PROGRAM MAIN
VAR
	pbGapMode: BOOL:=FALSE;
	pbTaperMode: BOOL:=FALSE;
	pbSingleCarrierMode: BOOL:=FALSE;
	pbDebugMode:BOOL:=FALSE;
	pbBCGapMode:BOOL:=FALSE;
	fb_led_Show: FB_LedShow;
	btn_reset: BOOL;
	CPMU_PLC_Reset: PLC_Reset;
	d_state: DINT;
	CPMU_PLC_Start: PLC_Start;
	powerStatus:BOOL;

(*TwinSAFE*)
	Safe_run AT%Q*:BOOL;
	Err_Ack AT %Q*:BOOL;
	Estop_RunAndRestart AT %Q*:BOOL;
	AX5805_Error_Ack AT %Q*:BOOL;
	Led_Run  AT %Q*:BOOL;
	Led_Error  AT %Q*:BOOL;

	FB_ERROR AT%I*:BOOL;
	COM_ERROR AT%I*:BOOL;
	//OUT_ERROR AT%I*:BOOL;
	Estop_Out AT%I*:BOOL;

	SafeStatus:INT;
	SafePLCRunOK: BOOL;
	fb_ton: TON;
	fb_ton2: TON;
	fb_ton3: TON;
	fb_ton1: TON;
	fb_ton0: TON;
(*IO*)
	el1808_D1  AT%I* :ARRAY[1..12] OF BOOL;
	el1808_D2  AT%I* :ARRAY[1..4] OF BOOL;
	el1008 AT%I*:BOOL;
	EStopTrig:BOOL;
(*setAxisPosition*)
	SetAxisPosState: INT;
	FB_Set_AxisPosition:FB_SetAxisPosition;
	fb_ton4: TON;
	fb_ton5: TON;
	fb_ton6: TON;
	SetAxisPositionDone: BOOL;
	//
	SetPhaseUpperAxisPosState: INT;
	FB_Set_PhaseUpperAxisPosition:FB_SetPhaseUpperAxisPosition;
	fb_ton7: TON;
	fb_ton8: TON;
	fb_ton9: TON;
	SetPhaseUpperAxisPositionDone: BOOL;
	//
	SetPhaseLowerAxisPosState: INT;
	FB_Set_PhaseLowerAxisPosition:FB_SetPhaseLowerAxisPosition;
	fb_ton10: TON;
	fb_ton11: TON;
	fb_ton12: TON;
	SetPhaseLowerAxisPositionDone: BOOL;
	i: INT;
	j: INT;

(****RS232***)
	fbEL6001	: FB_SerialCom;
	moveDoneLeftTop: BOOL;
	moveDoneRightTop: BOOL;
	moveDoneLeftBottom: BOOL;
	moveDoneRightBottom: BOOL;

(*Torque*)
	Torque_LT AT%I*:INT;
	Torque_RT AT%I*:INT;
	Torque_LB AT%I*:INT;
	Torque_RB AT%I*:INT;
	Torque_PU AT%I*:INT;
	Torque_PL AT%I*:INT;
(**)
	btn_setAxisPosition: BOOL;
	ValueSet_LeftTop:LREAL;
	ValueSet_RightTop:LREAL;
	ValueSet_LeftBottom:LREAL;
	ValueSet_RightBottom:LREAL;
	btn_setPhaseUpperAxisPosition: BOOL;
	PhaseUpperSetValue: LREAL;
	btn_setPhaseLowerAxisPosition: BOOL;
	PhaseLowerSetValue: LREAL;
(**)
	RestartTC: TC_Restart;
	
(*recipe*)
	RecipeINT:INT;
	RecipeBOOL:BOOL;
	RecipeManCommands: RecipeManCommands;
	SaveParameter : BOOL;  //保存文件
	LoadParameter : BOOL;  //读取文件
	Save_R_TRIG   : R_TRIG;
	Read_R_TRIG   : R_TRIG;
	loadparameterStatus: INT;
	RecipeBOOL2:BOOL;
	ReturnDwordLoad: DWORD;
	InsertionDeviceName:STRING;
(*UserMode*)
	pbUserMode: BOOL:=TRUE;
	EL1904 AT%I* :ARRAY[1..32] OF BOOL;
	setAxisPositionEnable: BOOL;
	setPhaseUpperAxisPositionEnable: BOOL;
	setPhaseLowerAxisPositionEnable: BOOL;
	state_loadParameters: INT;
	state_setLEPosBias: INT;
	//
	PositionBiasSet:BOOL;
	MC_SetLEPosBias_LeftTop:MC_WriteParameter;
	MC_SetLEPosBias_RightTop:MC_WriteParameter;
	MC_SetLEPosBias_LeftBottom:MC_WriteParameter;
	MC_SetLEPosBias_RightBottom:MC_WriteParameter;
	MC_SetLEPosBias_PhaseUpper:MC_WriteParameter;
	MC_SetLEPosBias_PhaseLower:MC_WriteParameter;
	PositionBias_LeftTop: LREAL:=10.1;
	PositionBias_RightTop: LREAL:=10.2;
	PositionBias_LeftBottom: LREAL:=10.3;
	PositionBias_RightBottom: LREAL:=10.4;
	PositionBias_PhaseUpper: LREAL:=10.3;
	PositionBias_PhaseLower: LREAL:=10.4;
	
	LoadLEPB_R_TRIG: R_TRIG;
	PositionBiasTON: TON;
	
	//
	OPC_TEST_Bi:BOOL:=TRUE; (*~ (OPC:1:available for OPC Clients) *)
	OPC_TEST_Bi2:BOOL;(*~ (OPC:1:available for OPC Clients) *)
	//
	HasTemperatureSensorOrNot:BOOL;//Only IVU or CPMU
	(*Sensor Reading*)
	Sensor_Reading_1 AT %I*:ARRAY[0..3] OF BYTE;
	Sensor_Reading_2 AT %I*:ARRAY[0..3] OF BYTE;
	Sensor_Reading_3 AT %I*:ARRAY[0..3] OF BYTE;
	Sensor_Reading_4 AT %I*:ARRAY[0..3] OF BYTE;
	Sensor_Reading_5 AT %I*:ARRAY[0..3] OF BYTE;
	Sensor_Reading_6 AT %I*:ARRAY[0..3] OF BYTE;
	Sensor_Reading_7 AT %I*:ARRAY[0..3] OF BYTE;
	Sensor_Reading_8 AT %I*:ARRAY[0..3] OF BYTE;
	Sensor_Reading_DpState AT %I*:USINT;
	Sensor_Reading_ExtDiagFlag AT %I*:BOOL;
	TemperatureSensors_1:LREAL;
	TemperatureSensors_2:LREAL;
	TemperatureSensors_3:LREAL;
	TemperatureSensors_4:LREAL;
	TemperatureSensors_5:LREAL;
	TemperatureSensors_6:LREAL;
	TemperatureSensors_7:LREAL;
	TemperatureSensors_8:LREAL;
	dut_sensor_datas_1:DUT_SENSOR_DATAS_1;
	dut_sensor_datas_2:DUT_SENSOR_DATAS_2;
	dut_sensor_datas_3:DUT_SENSOR_DATAS_3;
	dut_sensor_datas_4:DUT_SENSOR_DATAS_4;
	dut_sensor_datas_5:DUT_SENSOR_DATAS_5;
	dut_sensor_datas_6:DUT_SENSOR_DATAS_6;
	dut_sensor_datas_7:DUT_SENSOR_DATAS_7;
	dut_sensor_datas_8:DUT_SENSOR_DATAS_8;
	//
	temperature_gradient_2_To_1:LREAL;
	temperature_gradient_3_To_2:LREAL;
	temperature_gradient_5_To_4:LREAL;
	temperature_gradient_6_To_5:LREAL;
	temperature_gradient_max:LREAL;
	//
	temperature_average:LREAL;
	A_SetLinearEncoderPositionBias_Enable: BOOL;
	
		//
	temperatureStatus:INT;//0：有传感器度数错误；1:常温；2:低温；3:常温和低温中间态
	CryogenicTemperatureThreshold:LREAL:=80;//80K以下归划分为低温
	RoomTemperatureThreshold:LREAL:=293;//293K以上划分为常温
	//CPMU cryogenix ON/FF
	CryogenicCompensationOn:BOOL;
	CryogenicCompensationConditionsReady:BOOL;
	CryogenicCompensation_LeftTop:LREAL;
	CryogenicCompensation_RightTop:LREAL;
	CryogenicCompensation_LeftBottom:LREAL;
	CryogenicCompensation_RightBottom:LREAL;
	CryogenicCompensationDone: BOOL;
	
	(**)
	bDriveDiagMessageAndNumber  : BOOL;
	m_GetDriveStatusState:INT;
	GetDriveStatusStateDone:BOOL;
	GetDriveStatusStateError:BOOL;
	//	
	fb_SoEReadDiagMessage_LeftTop: FB_SoEReadDiagMessage;
	fb_SoEReadDiagMessage_RightTop: FB_SoEReadDiagMessage;
	fb_SoEReadDiagMessage_LeftBottom: FB_SoEReadDiagMessage;
	fb_SoEReadDiagMessage_RightBottom: FB_SoEReadDiagMessage;
	fb_SoEReadDiagMessage_PhaseUpper: FB_SoEReadDiagMessage;
	fb_SoEReadDiagMessage_PhaseLower: FB_SoEReadDiagMessage;
	DriveDiagMessage_LeftTop:STRING;
	DriveDiagMessage_RightTop:STRING;
	DriveDiagMessage_LeftBottom:STRING;
	DriveDiagMessage_RightBottom:STRING;
	DriveDiagMessage_PhaseUpper:STRING;
	DriveDiagMessage_PhaseLower:STRING;
	//
	FB_SoEReadDiagNumber_LeftTop: FB_SoEReadDiagNumber;
	FB_SoEReadDiagNumber_RightTop: FB_SoEReadDiagNumber;
	FB_SoEReadDiagNumber_LeftBottom: FB_SoEReadDiagNumber;
	FB_SoEReadDiagNumber_RightBottom: FB_SoEReadDiagNumber;
	FB_SoEReadDiagNumber_PhaseUpper: FB_SoEReadDiagNumber;
	FB_SoEReadDiagNumber_PhaseLower: FB_SoEReadDiagNumber;
	DriveDiagNumber_LeftTop:UDINT;
	DriveDiagNumber_RightTop:UDINT;
	DriveDiagNumber_LeftBottom:UDINT;
	DriveDiagNumber_RightBottom:UDINT;
	DriveDiagNumber_PhaseUpper:UDINT;
	DriveDiagNumber_PhaseLower:UDINT;
	bReloadDriveDiagMessageAndNumber: BOOL;
	
	(*load IOC*)
	bExe_load_Prog: BOOL;
	NT_StartProcess_Load: NT_StartProcess;
	Exe_load_step: UINT;
	R_TRIG_ExeLoad: R_TRIG;
	Exe_Load_Done:BOOL;
	(*kill IOC*)
	bExe_Kill_Prog: BOOL;
	NT_StartProcess_Kill: NT_StartProcess;
	Exe_kill_step: UINT;
	R_TRIG_Exekill: R_TRIG;
	Exe_Kill_Done:BOOL;
	LoadOpcIocTON:TON;
	
	GetDriveStatusTON:TON;
	
	//
	//more parameters get:gear;feedback2 direction 
	//
	//GetMoreDriveStatus_FunctionON:BOOL:=TRUE;
	GetDriveStatusTON2: TON;
	//GearNumerator,st182
	st_p182_LeftTop:ST_P182;
	FB_SoERead_GearNumerator_LeftTop: FB_SoERead;
	st_p182_RightTop:ST_P182;
	FB_SoERead_GearNumerator_RightTop: FB_SoERead;
	st_p182_LeftBottom:ST_P182;
	FB_SoERead_GearNumerator_LeftBottom: FB_SoERead;
	st_p182_RightBottom:ST_P182;
	FB_SoERead_GearNumerator_RightBottom: FB_SoERead;
	st_p182_PhaseUpper:ST_P182;
	FB_SoERead_GearNumerator_PhaseUpper: FB_SoERead;
	st_p182_PhaseLower:ST_P182;
	FB_SoERead_GearNumerator_PhaseLower: FB_SoERead;
	GearNumeratorGet_LeftTop:UDINT;
	GearNumeratorGet_RightTop:UDINT;
	GearNumeratorGet_LeftBottom:UDINT;
	GearNumeratorGet_RightBottom:UDINT;
	GearNumeratorGet_PhaseUpper:UDINT;
	GearNumeratorGet_PhaseLower:UDINT;
	GearNumeratorConfigured_LeftTop:UDINT;
	GearNumeratorConfigured_RightTop:UDINT;
	GearNumeratorConfigured_LeftBottom:UDINT;
	GearNumeratorConfigured_RightBottom:UDINT;
	GearNumeratorConfigured_PhaseUpper:UDINT;
	GearNumeratorConfigured_PhaseLower:UDINT;
	//GearDenominator,st183
	st_p183_LeftTop:ST_P183;
	FB_SoERead_GearDenominator_LeftTop: FB_SoERead;
	st_p183_RightTop:ST_P183;
	FB_SoERead_GearDenominator_RightTop: FB_SoERead;
	st_p183_LeftBottom:ST_P183;
	FB_SoERead_GearDenominator_LeftBottom: FB_SoERead;
	st_p183_RightBottom:ST_P183;
	FB_SoERead_GearDenominator_RightBottom: FB_SoERead;
	st_p183_PhaseUpper:ST_P183;
	FB_SoERead_GearDenominator_PhaseUpper: FB_SoERead;
	st_p183_PhaseLower:ST_P183;
	FB_SoERead_GearDenominator_PhaseLower: FB_SoERead;
	GearDenominatorGet_LeftTop:UDINT;
	GearDenominatorGet_RightTop:UDINT;
	GearDenominatorGet_LeftBottom:UDINT;
	GearDenominatorGet_RightBottom:UDINT;
	GearDenominatorGet_PhaseUpper:UDINT;
	GearDenominatorGet_PhaseLower:UDINT;
	GearDenominatorConfigured_LeftTop:UDINT;
	GearDenominatorConfigured_RightTop:UDINT;
	GearDenominatorConfigured_LeftBottom:UDINT;
	GearDenominatorConfigured_RightBottom:UDINT;
	GearDenominatorConfigured_PhaseUpper:UDINT;
	GearDenominatorConfigured_PhaseLower:UDINT;
	//Feedback2direction,st180
	st_p180_LeftTop:ST_P180;
	FB_SoERead_Feedback2direction_LeftTop: FB_SoERead;
	st_p180_RightTop:ST_P180;
	FB_SoERead_Feedback2direction_RightTop: FB_SoERead;
	st_p180_LeftBottom:ST_P180;
	FB_SoERead_Feedback2direction_LeftBottom: FB_SoERead;
	st_p180_RightBottom:ST_P180;
	FB_SoERead_Feedback2direction_RightBottom: FB_SoERead;
	st_p180_PhaseUpper:ST_P180;
	FB_SoERead_Feedback2direction_PhaseUpper: FB_SoERead;
	st_p180_PhaseLower:ST_P180;
	FB_SoERead_Feedback2direction_PhaseLower: FB_SoERead;
	Feedback2directionGet_LeftTop:UINT;
	Feedback2directionGet_RightTop:UINT;
	Feedback2directionGet_LeftBottom:UINT;
	Feedback2directionGet_RightBottom:UINT;
	Feedback2directionGet_PhaseUpper:UINT;
	Feedback2directionGet_PhaseLower:UINT;
	Feedback2directionConfigured_LeftTop:UINT;
	Feedback2directionConfigured_RightTop:UINT;
	Feedback2directionConfigured_LeftBottom:UINT;
	Feedback2directionConfigured_RightBottom:UINT;
	Feedback2directionConfigured_PhaseUpper:UINT;
	Feedback2directionConfigured_PhaseLower:UINT;
	
	//RestartDrivers
		(*重启驱动器*)
	btn_RestartDriversAll:BOOL;
	btn_RestartDriver1:BOOL;
	btn_RestartDriver2:BOOL;
	btn_RestartDriver3:BOOL;
	btn_RestartDriver4:BOOL;
	btn_RestartDriver5:BOOL;
	btn_RestartDriver6:BOOL;
	btn_RestartDriver7:BOOL;
	btn_RestartDriver8:BOOL;
	Relay_EL2624 AT %Q*:ARRAY[0..7]OF  BOOL;
	RestartDriver_RTRIG:R_TRIG;
	RestartDriver_TON:TON;
	RestartDriver_Triggered:BOOL;
	RestartDriver_State:DINT;
	RestartDriver_Done:BOOL;
	//
	
	//
	//	LEHeartBeatMonitorFunction
	//
	LEHeartBeatMonitorFunctionOn: BOOL;
	LEHeartBeatFirstScan:BOOL;
	LEHeartBeatDeadZone : LREAL := 0; 
	LEHeartBeatAlarmTime : TIME := T#0.1S;
	
    //Pos_LeftTopLin_Last : LREAL; 
	Velo_LeftTopLin_Last : LREAL; 
	Pos_LeftTopMotor_Initial : LREAL; 
    StableTimer_LeftTopLin : TON; 
    StableTime_LeftTopLin : TIME; 
    DeltaVelo_LeftTopLin : LREAL; 
	IsInitialPositionSet_LeftTop: BOOL;
	MotorPosChange_LeftTop: LREAL;
	Threshold_LeftTopMotorPos:LREAL:=0.1;
	Threshold_LeftTopMotorVelo:LREAL:=0.2;
	Alarm_LeftTopLin:BOOL;
	Alarm_LeftTopMotorPos:BOOL;
	Alarm_LeftTopMotorVelo:BOOL;
	
	
	//Pos_RightTopLin_Last : LREAL; 
	Velo_RightTopLin_Last : LREAL; 
	Pos_RightTopMotor_Initial : LREAL; 
    StableTimer_RightTopLin : TON; 
    StableTime_RightTopLin : TIME; 
    DeltaVelo_RightTopLin : LREAL; 
	IsInitialPositionSet_RightTop: BOOL;
	MotorPosChange_RightTop: LREAL; 
	Threshold_RightTopMotorPos:LREAL:=0.1;
	Threshold_RightTopMotorVelo:LREAL:=0.2;
	Alarm_RightTopLin:BOOL;
	Alarm_RightTopMotorPos:BOOL;
	Alarm_RightTopMotorVelo:BOOL;
	
		
    //Pos_LeftBottomLin_Last : LREAL; 
	Velo_LeftBottomLin_Last : LREAL; 
	Pos_LeftBottomMotor_Initial : LREAL; 
    StableTimer_LeftBottomLin : TON; 
    StableTime_LeftBottomLin : TIME; 
    DeltaVelo_LeftBottomLin : LREAL; 
	IsInitialPositionSet_LeftBottom: BOOL;
	MotorPosChange_LeftBottom: LREAL; 
	Threshold_LeftBottomMotorPos:LREAL:=0.1;
	Threshold_LeftBottomMotorVelo:LREAL:=0.2;
	Alarm_LeftBottomLin:BOOL;
	Alarm_LeftBottomMotorPos:BOOL;
	Alarm_LeftBottomMotorVelo:BOOL;
	
	//Pos_RightBottomLin_Last : LREAL; 
	Velo_RightBottomLin_Last : LREAL; 
	Pos_RightBottomMotor_Initial : LREAL; 
    StableTimer_RightBottomLin : TON; 
    StableTime_RightBottomLin : TIME; 
    DeltaVelo_RightBottomLin : LREAL; 
	IsInitialPositionSet_RightBottom: BOOL;
	MotorPosChange_RightBottom: LREAL; 
	Threshold_RightBottomMotorPos:LREAL:=0.1;
	Threshold_RightBottomMotorVelo:LREAL:=0.2;
	Alarm_RightBottomLin:BOOL;
	Alarm_RightBottomMotorPos:BOOL;
	Alarm_RightBottomMotorVelo:BOOL;
	
	//Pos_PhaseUpperLin_Last : LREAL; 
	Velo_PhaseUpperLin_Last : LREAL; 
	Pos_PhaseUpperMotor_Initial : LREAL; 
    StableTimer_PhaseUpperLin : TON; 
    StableTime_PhaseUpperLin : TIME; 
    DeltaVelo_PhaseUpperLin : LREAL; 
	IsInitialPositionSet_PhaseUpper: BOOL;
	MotorPosChange_PhaseUpper: LREAL; 
	Threshold_PhaseUpperMotorPos:LREAL:=0.1;
	Threshold_PhaseUpperMotorVelo:LREAL:=0.2;
	Alarm_PhaseUpperLin:BOOL;
	Alarm_PhaseUpperMotorPos:BOOL;
	Alarm_PhaseUpperMotorVelo:BOOL;
	
	//Pos_PhaseLowerLin_Last : LREAL; 
	Velo_PhaseLowerLin_Last : LREAL; 
	Pos_PhaseLowerMotor_Initial : LREAL; 
    StableTimer_PhaseLowerLin : TON; 
    StableTime_PhaseLowerLin : TIME; 
    DeltaVelo_PhaseLowerLin : LREAL; 
	IsInitialPositionSet_PhaseLower: BOOL;
	MotorPosChange_PhaseLower: LREAL; 
	Threshold_PhaseLowerMotorPos:LREAL:=0.1;
	Threshold_PhaseLowerMotorVelo:LREAL:=0.2;
	Alarm_PhaseLowerLin:BOOL;
	Alarm_PhaseLowerMotorPos:BOOL;
	Alarm_PhaseLowerMotorVelo:BOOL;
	
	(*setAxisPosition*)
	SetMotorAxisPosState: INT;
	FB_Set_MotorAxisPosition:FB_SetMotorAxisPosition;
	fb_ton4_2: TON;
	fb_ton5_2: TON;
	SetMotorAxisPositionDone: BOOL;
	btn_SetMotorAxisPosition: BOOL;	
	(*setAxisPosition-PhaseUpper*)
	SetPhaseUpperMotorAxisPosState: INT;
	FB_Set_PhaseUpperMotorAxisPosition:FB_SetPhaseUpperMotorAxisPosition;
	fb_ton7_2: TON;
	SetPhaseUpperMotorAxisPositionDone: BOOL;
	btn_SetPhaseUpperMotorAxisPosition: BOOL;
	(*setAxisPosition-PhaseLower*)
	SetPhaseLowerMotorAxisPosState: INT;
	FB_Set_PhaseLowerMotorAxisPosition:FB_SetPhaseLowerMotorAxisPosition;
	fb_ton8_2: TON;
	SetPhaseLowerMotorAxisPositionDone: BOOL;
	btn_SetPhaseLowerMotorAxisPosition: BOOL;
	
	
	MonitorMotorAndLEFunctionOn:BOOL:=TRUE;
	
		(*GetMotorTempture*)
	MotorTemperature AT %I*:ARRAY[0..5] OF UINT;
	MotorTemperature_LeftTop:LREAL;
	MotorTemperature_RightTop:LREAL;
	MotorTemperature_LeftBottom:LREAL;
	MotorTemperature_RightBottom:LREAL;
	MotorTemperature_PhaseUpper:LREAL;
	MotorTemperature_PhaseLower:LREAL;

	fbPolar    : FB_PolarizationState;
    stPolarizationParam   : ST_PolarizationParam;
END_VAR

(*MaintenanceMode*)
IF MaintenanceMode THEN
	MaintenanceModeLed:=TRUE;
	RETURN;
ELSE
	MaintenanceModeLed:=FALSE;	
END_IF
(*加载Ricipe参数*)
A_InitRecipeParameters();
(*Restart TwinCAT*)
IF Global_Variables.m_restartTC THEN
(*首先关闭opcIocShell.exe*)	
	bExe_Kill_Prog:=TRUE;
	A_KillOpcIocShellExe();
(*重启TC*)
	IF Exe_Kill_Done THEN
		A_RestartTC();
	END_IF
END_IF
(*******InitAxisParameters*******)
A_InitAxisParameters();
(*******¼à²âÏÞÎ»¿ª¹Ø×´Ì¬£¬·½Ïò¿ØÖÆ&½ô¼±Çé¿öÏÂEStop*******)
A_CheckLimitSwitch();
(*Check Kill Switch*)
A_CheckKillSwitch();
(*******PosDiff¼à¿Ø*******)
A_PosDiffDetectiion();
(*******³õÊ¼»¯SafePlc*******)
IF NOT simulation THEN
A_SafePlcStartInit();
END_IF
(************SetAxisPosition-GAP*********************)
IF  NOT USELinearEncoder AND setAxisPositionEnable AND btn_setAxisPosition THEN
		FB_Set_AxisPosition.ValueSet_LeftTop:=ValueSet_LeftTop;
		FB_Set_AxisPosition.ValueSet_RightTop:=ValueSet_RightTop;
		FB_Set_AxisPosition.ValueSet_LeftBottom:=ValueSet_LeftBottom;
		FB_Set_AxisPosition.ValueSet_RightBottom:=ValueSet_RightBottom;
		A_SetAxisPosition();
END_IF
(************SetAxisPosition-GAP*********************)
IF  NOT USELinearEncoder AND setPhaseUpperAxisPositionEnable AND btn_setPhaseUpperAxisPosition THEN
		FB_Set_PhaseUpperAxisPosition.ValueSet:=PhaseUpperSetValue;
		A_SetPhaseUpperAxisPosition();
END_IF
(************SetAxisPosition-GAP*********************)
IF  NOT USELinearEncoder AND setPhaseLowerAxisPositionEnable AND btn_setPhaseLowerAxisPosition THEN
		FB_Set_PhaseLowerAxisPosition.ValueSet:=PhaseLowerSetValue;
		A_SetPhaseLowerAxisPosition();
END_IF
(*******模式选择******)
IF SafePLCRunOK OR Simulation THEN
	IF pbSingleCarrierMode AND NOT pbTaperMode AND NOT pbGapMode AND NOT pbDebugMode AND NOT pbBCGapMode AND NOT pbUserMode THEN
		SingleCarrierMode();
	ELSIF pbTaperMode  AND NOT pbSingleCarrierMode AND NOT pbGapMode  AND NOT pbDebugMode AND NOT pbBCGapMode AND NOT pbUserMode THEN
		TaperMode();
	ELSIF pbGapMode AND  NOT pbSingleCarrierMode AND NOT pbTaperMode  AND NOT pbDebugMode AND NOT pbBCGapMode AND NOT pbUserMode THEN
		GapMode();
	ELSIF pbDebugMode AND NOT pbGapMode AND NOT pbSingleCarrierMode AND NOT pbTaperMode AND NOT pbBCGapMode  AND NOT pbUserMode THEN
		DebugMode();
	ELSIF pbBCGapMode AND NOT pbGapMode AND NOT pbSingleCarrierMode AND NOT pbTaperMode AND NOT pbDebugMode AND NOT pbUserMode THEN
		BCGapMode();
	ELSIF pbUserMode AND NOT pbGapMode AND NOT pbSingleCarrierMode AND NOT pbTaperMode AND NOT pbDebugMode AND NOT pbBCGapMode THEN
		UserMode();
	END_IF
END_IF
(*******Led Show******)
fb_led_Show();
(*******Check Power status******)
FB_Power(Check:=TRUE);
st_Power:=FB_Power.PowerState;
(******Check Couple Status*****)
FB_CheckCoupleStatus(Check:=TRUE);
st_Couple:=FB_CheckCoupleStatus.CoupleState;

(*********RS232*********************)
BackgroundEL();

(*获取温度传感器数据*)
//A_GetTemperatureSensorsData();

(*设置position bias*)
IF loadParametersDone AND (DriveStatus=1 OR simulation) THEN 
	A_SetLinearEncoderPositionBias();
END_IF
(*检查硬急停状态，包括安全限位、柜门急停、手持急停*)
A_CheckHardwareEmergencyStopStatus();
IF NOT simulation THEN
	A_GetDriverStatus();
END_IF
(*IDControlReady*)
IF ((DriveStatus<>0 AND SafePLCRunOK) OR simulation) AND NOT Error THEN
	IDControlReady:=TRUE;
ELSE
	IDControlReady:=FALSE;
END_IF

(*IOC Start*)
IF SafePLCRunOK OR simulation THEN
	bExe_load_Prog:=TRUE;
	A_LoadOpcIocShellExe();
END_IF

(*RestartDrivers*)
A_RestartDrivers();

(*检查光栅读数是否在范围内*)
A_CheckLinearEncoder();


(*A_LEHeartBeatMonitor*)
IF LEHeartBeatMonitorFunctionOn THEN
	A_LEHeartBeatMonitor();
END_IF
(************SetMotorAxisPosition*********************)
//IDControl 1s after
fb_ton5_2.IN:=IDControlReady;
fb_ton5_2.PT:=T#1S;
fb_ton5_2();
IF fb_ton5_2.Q THEN
	btn_SetMotorAxisPosition:=TRUE;
	btn_SetPhaseUpperMotorAxisPosition:=TRUE;
	btn_SetPhaseLowerMotorAxisPosition:=TRUE;
END_IF
IF  USELinearEncoder AND btn_SetMotorAxisPosition THEN
	IF NOT SetMotorAxisPositionDone THEN
		FB_Set_MotorAxisPosition.ValueSet_LeftTop:=Pos_LeftTopLin;
		FB_Set_MotorAxisPosition.ValueSet_RightTop:=Pos_RightTopLin;
		FB_Set_MotorAxisPosition.ValueSet_LeftBottom:=Pos_LeftBottomLin;
		FB_Set_MotorAxisPosition.ValueSet_RightBottom:=Pos_RightBottomLin;
		A_SetMotorAxisPosition();
	END_IF
END_IF
IF  USELinearEncoder AND btn_SetPhaseUpperMotorAxisPosition THEN
	IF NOT SetPhaseUpperMotorAxisPositionDone THEN
		FB_Set_PhaseUpperMotorAxisPosition.ValueSet:=Pos_PhaseUpperLin;
		A_SetPhaseUpperMotorAxisPosition();
	END_IF
END_IF
IF  USELinearEncoder AND btn_SetPhaseLowerMotorAxisPosition THEN
	IF NOT SetPhaseLowerMotorAxisPositionDone THEN
		FB_Set_PhaseLowerMotorAxisPosition.ValueSet:=Pos_PhaseLowerLin;
		A_SetPhaseLowerMotorAxisPosition();
	END_IF
END_IF
(*A_MonitorMotorAndLE*)
IF MonitorMotorAndLEFunctionOn AND SetMotorAxisPositionDone 
	AND SetPhaseUpperMotorAxisPositionDone AND SetPhaseLowerMotorAxisPositionDone THEN
	A_MonitorMotorAndLE();
END_IF
(*A_CheckMaxVelocity*)
A_CheckMaxVelocity();
(**)
A_GetMotorTemperature();

A_PolarStatus();

ACTION A_CheckHardwareEmergencyStopStatus:
IF 	NOT KS_LeftTop_Far_Contact1 OR
	NOT KS_LeftTop_Far_Contact2 OR
	NOT KS_RightTop_Far_Contact1 OR
	NOT KS_RightTop_Far_Contact2 OR
	NOT KS_LeftBottom_Far_Contact1 OR
	NOT KS_LeftBottom_Far_Contact2 OR
	NOT KS_RightBottom_Far_Contact1 OR
	NOT KS_RightBottom_Far_Contact2 OR
	NOT KS_PhaseUpper_Exit_Contact1 OR
	NOT KS_PhaseUpper_Exit_Contact2 OR
	NOT KS_PhaseLower_Exit_Contact1 OR
	NOT KS_PhaseLower_Exit_Contact2 OR
	
	NOT KS_LeftTop_Near_Contact1 OR
	NOT KS_LeftTop_Near_Contact2 OR
	NOT KS_RightTop_Near_Contact1 OR
	NOT KS_RightTop_Near_Contact2 OR
	NOT KS_LeftBottom_Near_Contact1 OR
	NOT KS_LeftBottom_Near_Contact2 OR
	NOT KS_RightBottom_Near_Contact1 OR
	NOT KS_RightBottom_Near_Contact2 OR
	NOT KS_PhaseUpper_Entrance_Contact1 OR
	NOT KS_PhaseUpper_Entrance_Contact2 OR
	NOT KS_PhaseLower_Entrance_Contact1 OR
	NOT KS_PhaseLower_Entrance_Contact2 OR
(*E-STOP*)
	NOT KS_CabinetEmergency_contact1 OR
	NOT KS_CabinetEmergency_contact2 OR
	NOT KS_handEmergency1_Contact1 OR
	NOT KS_handEmergency1_Contact2 OR
	NOT KS_handEmergency2_Contact1 OR
	NOT KS_handEmergency2_Contact2 OR
	NOT KS_softEmergency2_Contact THEN
	Hardware_EmergencyStop:=FALSE;
ELSE
	Hardware_EmergencyStop:=TRUE;
END_IF
END_ACTION

ACTION A_CheckKillSwitch:
IF simulation THEN
	//EL1904-1
	KS_LeftTop_Far_Contact1:=TRUE;
	KS_LeftTop_Far_Contact2:=TRUE;
	KS_LeftTop_Near_Contact1:=TRUE;
	KS_LeftTop_Near_Contact2:=TRUE;
	//EL1904-2
	KS_RightTop_Far_Contact1:=TRUE;
	KS_RightTop_Far_Contact2:=TRUE;
	KS_RightTop_Near_Contact1:=TRUE;
	KS_RightTop_Near_Contact2:=TRUE;
	//EL1904-3
	KS_LeftBottom_Far_Contact1:=TRUE;
	KS_LeftBottom_Far_Contact2:=TRUE;
	KS_LeftBottom_Near_Contact1:=TRUE;
	KS_LeftBottom_Near_Contact2:=TRUE;
	//EL1904-4
	KS_RightBottom_Far_Contact1:=TRUE;
	KS_RightBottom_Far_Contact2:=TRUE;
	KS_RightBottom_Near_Contact1:=TRUE;
	KS_RightBottom_Near_Contact2:=TRUE;
	//EL1904-5
	KS_PhaseUpper_Exit_Contact1:=TRUE;
	KS_PhaseUpper_Exit_Contact2:=TRUE;
	KS_PhaseUpper_Entrance_Contact1:=TRUE;
	KS_PhaseUpper_Entrance_Contact2:=TRUE;
	//EL1904-6
	KS_PhaseLower_Exit_Contact1:=TRUE;
	KS_PhaseLower_Exit_Contact2:=TRUE;
	KS_PhaseLower_Entrance_Contact1:=TRUE;
	KS_PhaseLower_Entrance_Contact2:=TRUE;
	//EL1904-7
	(*E-STOP*)
	(*柜门急停*)
	KS_CabinetEmergency_contact1:=TRUE;
	KS_CabinetEmergency_contact2:=TRUE;
	(*手持急停-1*)
	KS_handEmergency1_Contact1:=TRUE;
	KS_handEmergency1_Contact2:=TRUE;
	//EL1904-8
	(*手持急停-2*)
	KS_handEmergency2_Contact1:=TRUE;
	KS_handEmergency2_Contact2:=TRUE;
	
	KS_softEmergency2_Contact:=TRUE;
	AX5805_ErrorAsk:=TRUE;
ELSE
	//EL1904-1
	KS_LeftTop_Far_Contact1:=EL1904[1];//c1
	KS_LeftTop_Far_Contact2:=EL1904[2];//c2
	KS_LeftTop_Near_Contact1:=EL1904[3];//c3
	KS_LeftTop_Near_Contact2:=EL1904[4];//c4
	//EL1904-2
	KS_RightTop_Far_Contact1:=EL1904[5];
	KS_RightTop_Far_Contact2:=EL1904[6];
	KS_RightTop_Near_Contact1:=EL1904[7];
	KS_RightTop_Near_Contact2:=EL1904[8];
	//EL1904-3
	KS_LeftBottom_Far_Contact1:=EL1904[9];
	KS_LeftBottom_Far_Contact2:=EL1904[10];
	KS_LeftBottom_Near_Contact1:=EL1904[11];
	KS_LeftBottom_Near_Contact2:=EL1904[12];
	//EL1904-4
	KS_RightBottom_Far_Contact1:=EL1904[13];
	KS_RightBottom_Far_Contact2:=EL1904[14];
	KS_RightBottom_Near_Contact1:=EL1904[15];
	KS_RightBottom_Near_Contact2:=EL1904[16];	
	//EL1904-5
	KS_PhaseUpper_Exit_Contact1:=EL1904[17];
	KS_PhaseUpper_Exit_Contact2:=EL1904[18];
	KS_PhaseUpper_Entrance_Contact1:=EL1904[19];
	KS_PhaseUpper_Entrance_Contact2:=EL1904[20];
	//EL1904-6
	KS_PhaseLower_Exit_Contact1:=EL1904[21];
	KS_PhaseLower_Exit_Contact2:=EL1904[22];
	KS_PhaseLower_Entrance_Contact1:=EL1904[23];
	KS_PhaseLower_Entrance_Contact2:=EL1904[24];
	//EL1904-7
	(*E-STOP*)
	(*柜门急停*)
	KS_CabinetEmergency_contact1:=EL1904[25];
	KS_CabinetEmergency_contact2:=EL1904[26];
	(*手持急停-1*)
	KS_handEmergency1_Contact1:=EL1904[27];
	KS_handEmergency1_Contact2:=EL1904[28];
	//EL1904-8
	(*手持急停-2*)
	KS_handEmergency2_Contact1:=EL1904[29];
	KS_handEmergency2_Contact2:=EL1904[30];
	
	KS_softEmergency2_Contact:=EL1904[31];
	AX5805_ErrorAsk:=EL1904[32];

END_IF
END_ACTION

ACTION A_CheckLimitSwitch:
(*******1.´ÓIO»ñÈ¡ÏÞÎ»×´Ì¬******)
(**)

IF simulation THEN
	(**)
	LS_LeftTop_Far:=TRUE;
	LS_LeftTop_Near:=TRUE;
	LS_RightTop_Far:=TRUE;
	LS_RightTop_Near:=TRUE;
	LS_LeftBottom_Far:=TRUE;
	LS_LeftBottom_Near:=TRUE;
	LS_RightBottom_Far:=TRUE;
	LS_RightBottom_Near:=TRUE;
	LS_PhaseUpper_Entrance:=TRUE;
	LS_PhaseUpper_Exit:=TRUE;
	LS_PhaseLower_Entrance:=TRUE;
	LS_PhaseLower_Exit:=TRUE;
	
ELSE
	LS_LeftTop_Far :=el1808_D1[1];
	LS_LeftTop_Near:=el1808_D1[3];
	LS_RightTop_Far:=el1808_D1[2];
	LS_RightTop_Near:=el1808_D1[4];
	LS_LeftBottom_Far:=el1808_D1[7];
	LS_LeftBottom_Near:=el1808_D1[5];
	LS_RightBottom_Far:=el1808_D1[8];
	LS_RightBottom_Near:=el1808_D1[6];
	LS_PhaseUpper_Entrance:=el1808_D2[1];
	LS_PhaseUpper_Exit:=el1808_D2[2];
	LS_PhaseLower_Entrance:=el1808_D2[3];
	LS_PhaseLower_Exit:=el1808_D2[4];
END_IF


(*
	LS_LeftTop_Top:=TRUE;
	LS_LeftTop_Bottom:=TRUE;
	LS_RightTop_Top:=TRUE;
	LS_RightTop_Bottom:=TRUE;
	LS_LeftBottom_Top:=TRUE;
	LS_LeftBottom_Bottom:=TRUE;
	LS_RightBottom_Top:=TRUE;
	LS_RightBottom_Bottom:=TRUE;
*)
(******2.TopÏÞÎ»»òÕßBottomÏÞÎ»ÓÐÒ»¸ö´¥·¢£¬È«¾Ö±äÁ¿¡£¸øMC_POWERÓÃÓÚ·½Ïò¿ØÖÆ£¬ÓÐÒ»¸öÏÞÎ»Îª´¥·¢ÎªFALSE£¬ÔòUnreach_LSÎªFALSE******)
Unreach_LS_Far:=LS_LeftTop_Far AND LS_RightTop_Far AND LS_LeftBottom_Far AND LS_RightBottom_Far;
Unreach_LS_Near:=LS_LeftTop_Near AND LS_RightTop_Near AND LS_LeftBottom_Near AND LS_RightBottom_Near;
(**************************ÏòTopÔË¶¯Ê±£¬´¥ÅöBottomÏÞÎ»¿ª¹Ø£¬»òÕßÏà·´£¬ESTOP**************************************)
(*
IF LeftTopLin.Status.Moving AND Velo_LeftTopLin>0 THEN
	IF NOT Unreach_LS_Bottom THEN
		Error:=TRUE;
		ErrorID:=61;
		FB_PlcEmergencyStop();
	END_IF
ELSIF LeftTopLin.Status.Moving AND Velo_LeftTopLin<0 THEN
	IF NOT Unreach_LS_Top THEN
		Error:=TRUE;
		ErrorID:=62;
		FB_PlcEmergencyStop();
	END_IF
ELSIF RightTopLin.Status.Moving AND Velo_RightTopLin>0 THEN
	IF NOT Unreach_LS_Bottom THEN
		Error:=TRUE;
		ErrorID:=63;
		FB_PlcEmergencyStop();
	END_IF
ELSIF RightTopLin.Status.Moving AND Velo_RightTopLin<0 THEN
	IF NOT  Unreach_LS_Top THEN
		Error:=TRUE;
		ErrorID:=64;
		FB_PlcEmergencyStop();
	END_IF
ELSIF LeftBottomLin.Status.Moving AND Velo_LeftBottomLin>0 THEN
	IF NOT Unreach_LS_Bottom THEN
		Error:=TRUE;
		ErrorID:=65;
		FB_PlcEmergencyStop();
	END_IF
ELSIF LeftBottomLin.Status.Moving AND Velo_LeftBottomLin<0 THEN
	IF NOT Unreach_LS_Top THEN
		Error:=TRUE;
		ErrorID:=66;
		FB_PlcEmergencyStop();
	END_IF
ELSIF RightBottomLin.Status.Moving AND Velo_RightBottomLin>0 THEN
	IF NOT Unreach_LS_Bottom THEN
		Error:=TRUE;
		ErrorID:=67;
		FB_PlcEmergencyStop();
	END_IF
ELSIF RightBottomLin.Status.Moving AND Velo_RightBottomLin<0 THEN
	IF NOT Unreach_LS_Top THEN
		Error:=TRUE;
		ErrorID:=68;
		FB_PlcEmergencyStop();
	END_IF
END_IF
*)
(*
(******3.ÓÐÒ»¸öÏÞÎ»´¥·¢£¬ delayÊ±¼äºó£¬¼à²âÖáÊÇ·ñÔÚÍ£Ö¹×´Ì¬£¬ÈôÃ»ÓÐ£¬Emergency AND PowerOff******)
IF NOT Unreach_LS_Top OR NOT Unreach_LS_Bottom THEN
	fb_ton.IN:=TRUE;
END_IF
IF fb_ton.Q THEN
	IF LeftTopLin.Status.Moving OR RightTopLin.Status.Moving OR LeftBottomLin.Status.Moving OR RightBottomLin.Status.Moving THEN
		FB_PlcEmergencyStop();
		fb_ton.IN:=FALSE;
		Error:=TRUE;
		EStopTrig:=TRUE;
		ErrorID:=1;
		(*FB_Power_Off(Execute:=TRUE);*)
	END_IF
END_IF

(*******4.µ¥ÖáÉÏÏÂÏÞÎ»¾ùÎªFALSEÊ±£¬ÏÞÎ»´íÎó£¬Emergency*******)
IF (NOT LS_LeftTop_Top AND NOT LS_LeftTop_Bottom) OR  (NOT  LS_RightTop_Top AND NOT LS_RightTop_Bottom)
		OR (NOT LS_LeftBottom_Top AND NOT LS_LeftBottom_Bottom) OR (NOT LS_RightBottom_Top AND NOT LS_RightBottom_Bottom) THEN
	(*FB_Plc_EmergencyStop();*)
	Error:=TRUE;
	EStopTrig:=TRUE;
	ErrorID:=2;
END_IF
*)
END_ACTION

ACTION A_CheckLinearEncoder:
//LE Protection Position
min_UserLEProtectionGapPosition:=min_UserGapPositionNew-min_ThresholdGapSoft2LEProtection;//回程误差有0.1mm
max_UserLEProtectionGapPosition:=max_UserGapPositionNew+max_ThresholdGapSoft2LEProtection;
//如果没有使用光栅、或者光栅参数没设置好，则不检查光栅位置
IF NOT USELinearEncoder OR NOT PositionBiasDone THEN
	RETURN;
END_IF
IF Pos_LeftTopLin <=0 THEN
	ErrorID:=1101;
	Error:=TRUE;
	ErrorDescription:='Pos_LeftTopLin <=0';
	FB_PlcEmergencyStop();
	LED_Error:=TRUE;
END_IF
IF Pos_RightTopLin <=0 THEN
	ErrorID:=1102;
	Error:=TRUE;
	ErrorDescription:='Pos_RightTopLin <=0';
	FB_PlcEmergencyStop();
	LED_Error:=TRUE;
END_IF
IF Pos_LeftBottomLin <=0 THEN
	ErrorID:=1103;
	Error:=TRUE;
	ErrorDescription:='Pos_LeftBottomLin <=0';
	FB_PlcEmergencyStop();
	LED_Error:=TRUE;
END_IF
IF Pos_RightBottomLin <=0 THEN
	ErrorID:=1104;
	Error:=TRUE;
	ErrorDescription:='Pos_RightBottomLin <=0';
	FB_PlcEmergencyStop();
	LED_Error:=TRUE;
END_IF

//
IF Pos_LeftTopLin >max_UserLEProtectionGapPosition/2 THEN
	ErrorID:=1105;
	Error:=TRUE;
	ErrorDescription:='Pos_LeftTopLin >max_UserLEProtectionGapPosition/2';
	FB_PlcEmergencyStop();
	LED_Error:=TRUE;
END_IF
IF Pos_RightTopLin >max_UserLEProtectionGapPosition/2 THEN
	ErrorID:=1106;
	Error:=TRUE;
	ErrorDescription:='Pos_RightTopLin>max_UserLEProtectionGapPosition/2';
	FB_PlcEmergencyStop();
	LED_Error:=TRUE;
END_IF
IF Pos_LeftBottomLin >max_UserLEProtectionGapPosition/2 THEN
	ErrorID:=1107;
	Error:=TRUE;
	ErrorDescription:='Pos_LeftBottomLin >max_UserLEProtectionGapPosition/2';
	FB_PlcEmergencyStop();
	LED_Error:=TRUE;
END_IF
IF Pos_RightBottomLin >max_UserLEProtectionGapPosition/2 THEN
	ErrorID:=1108;
	Error:=TRUE;
	ErrorDescription:='Pos_RightBottomLin >max_UserLEProtectionGapPosition/2';
	FB_PlcEmergencyStop();
	LED_Error:=TRUE;
END_IF


IF Pos_LeftTopLin <min_UserLEProtectionGapPosition/2 THEN
	ErrorID:=1109;
	Error:=TRUE;
	ErrorDescription:='Pos_LeftTopLin <min_UserLEProtectionGapPosition/2';
	FB_PlcEmergencyStop();
	LED_Error:=TRUE;
END_IF
IF Pos_RightTopLin <min_UserLEProtectionGapPosition/2 THEN
	ErrorID:=1110;
	Error:=TRUE;
	ErrorDescription:='Pos_RightTopLin<min_UserLEProtectionGapPosition/2';
	FB_PlcEmergencyStop();
	LED_Error:=TRUE;
END_IF
IF Pos_LeftBottomLin <min_UserLEProtectionGapPosition/2 THEN
	ErrorID:=1111;
	Error:=TRUE;
	ErrorDescription:='Pos_LeftBottomLin <min_UserLEProtectionGapPosition';
	FB_PlcEmergencyStop();
	LED_Error:=TRUE;
END_IF
IF Pos_RightBottomLin <min_UserLEProtectionGapPosition/2 THEN
	ErrorID:=1112;
	Error:=TRUE;
	ErrorDescription:='Pos_RightBottomLin <min_UserLEProtectionGapPosition';
	FB_PlcEmergencyStop();
	LED_Error:=TRUE;
END_IF
//
//PhaseUpper方向
//
min_UserLEProtectionPhaseUpperPosition:=min_UserPhaseUpperPositionNew-min_ThresholdPhaseUpperSoft2LEProtection;//回程误差有0.1mm
max_UserLEProtectionPhaseUpperPosition:=max_UserPhaseUpperPositionNew+max_ThresholdPhaseUpperSoft2LEProtection;
IF Pos_PhaseUpperLin >max_UserLEProtectionPhaseUpperPosition THEN
	ErrorID:=1113;
	Error:=TRUE;
	ErrorDescription:=' Pos_PhaseUpperLin >max_UserLEProtectionPhaseUpperPosition';
	FB_PlcEmergencyStop();
	LED_Error:=TRUE;
END_IF
IF Pos_PhaseUpperLin < min_UserLEProtectionPhaseUpperPosition THEN
	ErrorID:=1114;
	Error:=TRUE;
	ErrorDescription:=' Pos_PhaseUpperLin >< min_UserLEProtectionPhaseUpperPosition';
	FB_PlcEmergencyStop();
	LED_Error:=TRUE;
END_IF
//
//PhaseLower方向
//
min_UserLEProtectionPhaseLowerPosition:=min_UserPhaseLowerPositionNew-min_ThresholdPhaseLowerSoft2LEProtection;//回程误差有0.1mm
max_UserLEProtectionPhaseLowerPosition:=max_UserPhaseLowerPositionNew+max_ThresholdPhaseLowerSoft2LEProtection;
IF Pos_PhaseLowerLin >max_UserLEProtectionPhaseLowerPosition THEN
	ErrorID:=1115;
	Error:=TRUE;
	ErrorDescription:=' Pos_PhaseLowerLin >max_UserLEProtectionPhaseLowerPosition';
	FB_PlcEmergencyStop();
	LED_Error:=TRUE;
END_IF
IF Pos_PhaseLowerLin < min_UserLEProtectionPhaseLowerPosition THEN
	ErrorID:=1116;
	Error:=TRUE;
	ErrorDescription:=' Pos_PhaseLowerLin < min_UserLEProtectionPhaseLowerPosition';
	FB_PlcEmergencyStop();
	LED_Error:=TRUE;
END_IF
END_ACTION

ACTION A_CheckMaxVelocity:
IF NOT USELinearEncoder OR NOT PositionBiasDone OR NOT IDControlReady THEN
	RETURN;
END_IF
IF NOT st_Power THEN
	RETURN;
END_IF
//Monitoring Motor and LE Position/Velocity
MaxVelocityGlobalVelocity:=MAX(max_UserGapVelocityNew,max_UserTaperVelocityNew,UserMode.max_SS_StepVelocity,
			UserMode.Global_ChainProtection_MPS_MoveVelocity,UserMode.Global_ChainProtection_EPS_MoveVelocity);
IF 	ABS(Velo_LeftTopLin) > MaxVelocityGlobalVelocity*1.1/2 THEN
	ErrorID:=7001;
	Error:=TRUE;
	ErrorDescription:='ABS(Velo_LeftTopLin) > MaxVelocityGlobalVelocity*1.1/2';
	FB_PlcEmergencyStop();
	LED_Error:=TRUE;
END_IF
IF 	ABS(Velo_LeftTopMotor) > MaxVelocityGlobalVelocity*1.1/2 THEN
	ErrorID:=7002;
	Error:=TRUE;
	ErrorDescription:='ABS(Velo_LeftTopMotor) > MaxVelocityGlobalVelocity*1.1/2';
	FB_PlcEmergencyStop();
	LED_Error:=TRUE;
END_IF
IF 	ABS(Velo_RightTopLin) > MaxVelocityGlobalVelocity*1.1/2 THEN
	ErrorID:=7003;
	Error:=TRUE;
	ErrorDescription:='ABS(Velo_RightTopLin) > MaxVelocityGlobalVelocity*1.1/2';
	FB_PlcEmergencyStop();
	LED_Error:=TRUE;
END_IF
IF 	ABS(Velo_RightTopMotor) > MaxVelocityGlobalVelocity*1.1/2 THEN
	ErrorID:=7004;
	Error:=TRUE;
	ErrorDescription:='ABS(Velo_RightTopMotor) > MaxVelocityGlobalVelocity*1.1/2';
	FB_PlcEmergencyStop();
	LED_Error:=TRUE;
END_IF
IF 	ABS(Velo_LeftBottomLin) > MaxVelocityGlobalVelocity*1.1/2 THEN
	ErrorID:=7005;
	Error:=TRUE;
	ErrorDescription:='ABS(Velo_LeftBottomLin) > MaxVelocityGlobalVelocity*1.1/2';
	FB_PlcEmergencyStop();
	LED_Error:=TRUE;
END_IF
IF 	ABS(Velo_LeftBottomMotor) > MaxVelocityGlobalVelocity*1.1/2 THEN
	ErrorID:=7006;
	Error:=TRUE;
	ErrorDescription:='ABS(Velo_LeftBottomMotor) > MaxVelocityGlobalVelocity*1.1/2';
	FB_PlcEmergencyStop();
	LED_Error:=TRUE;
END_IF
IF 	ABS(Velo_RightBottomLin) > MaxVelocityGlobalVelocity*1.1/2 THEN
	ErrorID:=7007;
	Error:=TRUE;
	ErrorDescription:='ABS(Velo_RightBottomLin) > MaxVelocityGlobalVelocity*1.1/2';
	FB_PlcEmergencyStop();
	LED_Error:=TRUE;
END_IF
IF 	ABS(Velo_RightBottomMotor) > MaxVelocityGlobalVelocity*1.1/2 THEN
	ErrorID:=7008;
	Error:=TRUE;
	ErrorDescription:='ABS(Velo_RighBottomMotor) > MaxVelocityGlobalVelocity*1.1/2';
	FB_PlcEmergencyStop();
	LED_Error:=TRUE;
END_IF
(*
IF 	ABS(Velo_PhaseUpperLin) > MaxVelocityGlobalVelocity*1.1/2 THEN
	ErrorID:=7005;
	Error:=TRUE;
	ErrorDescription:='ABS(Velo_PhaseUpperLin) > MaxVelocityGlobalVelocity*1.1/2';
	FB_PlcEmergencyStop();
	LED_Error:=TRUE;
END_IF
IF 	ABS(Velo_PhaseUpperMotor) > MaxVelocityGlobalVelocity*1.1/2 THEN
	ErrorID:=7006;
	Error:=TRUE;
	ErrorDescription:='ABS(Velo_PhaseUpperMotor) > MaxVelocityGlobalVelocity*1.1/2';
	FB_PlcEmergencyStop();
	LED_Error:=TRUE;
END_IF
IF 	ABS(Velo_PhaseLowerLin) > MaxVelocityGlobalVelocity*1.1/2 THEN
	ErrorID:=7007;
	Error:=TRUE;
	ErrorDescription:='ABS(Velo_PhaseLowerLin) > MaxVelocityGlobalVelocity*1.1/2';
	FB_PlcEmergencyStop();
	LED_Error:=TRUE;
END_IF
IF 	ABS(Velo_PhaseLowerMotor) > MaxVelocityGlobalVelocity*1.1/2 THEN
	ErrorID:=7008;
	Error:=TRUE;
	ErrorDescription:='ABS(Velo_RighBottomMotor) > MaxVelocityGlobalVelocity*1.1/2';
	FB_PlcEmergencyStop();
	LED_Error:=TRUE;
END_IF
*)
END_ACTION

ACTION A_GetDriverStatus:
//
//DriveMessage/Drive Number/Gear number/feedback2 direction
//
IF bReloadDriveDiagMessageAndNumber THEN
	m_GetDriveStatusState:=0;
	bReloadDriveDiagMessageAndNumber:=FALSE;
END_IF
GetDriveStatusTON(PT:=T#1S);
GetDriveStatusTON2(PT:=T#0.1S);
A_GetDriverStatusMC();
CASE m_GetDriveStatusState OF
	0:
		GetDriveStatusTON.IN:=TRUE;
		m_GetDriveStatusState:=1;
	1:
		IF GetDriveStatusTON.Q THEN
			bDriveDiagMessageAndNumber:=TRUE;
			m_GetDriveStatusState:=2;
		END_IF
	2:
		GetDriveStatusTON.IN:=FALSE;
		DriveDiagMessage_LeftTop:=fb_SoEReadDiagMessage_LeftTop.sDiagMessage.strData;
		DriveDiagMessage_RightTop:=fb_SoEReadDiagMessage_RightTop.sDiagMessage.strData;
		DriveDiagMessage_LeftBottom:=fb_SoEReadDiagMessage_LeftBottom.sDiagMessage.strData;
		DriveDiagMessage_RightBottom:=fb_SoEReadDiagMessage_RightBottom.sDiagMessage.strData;
		DriveDiagMessage_PhaseUpper:=fb_SoEReadDiagMessage_PhaseUpper.sDiagMessage.strData;
		DriveDiagMessage_PhaseLower:=fb_SoEReadDiagMessage_PhaseLower.sDiagMessage.strData;
		//
		DriveDiagNumber_LeftTop:=FB_SoEReadDiagNumber_LeftTop.iDiagNumber;
		DriveDiagNumber_RightTop:=FB_SoEReadDiagNumber_RightTop.iDiagNumber;
		DriveDiagNumber_LeftBottom:=FB_SoEReadDiagNumber_LeftBottom.iDiagNumber;
		DriveDiagNumber_RightBottom:=FB_SoEReadDiagNumber_RightBottom.iDiagNumber;
		DriveDiagNumber_PhaseUpper:=FB_SoEReadDiagNumber_PhaseUpper.iDiagNumber;
		DriveDiagNumber_PhaseLower:=FB_SoEReadDiagNumber_PhaseLower.iDiagNumber;
		//
		GearNumeratorGet_LeftTop:=st_p182_LeftTop.Feedback_2_geat_numerator;
		GearNumeratorGet_RightTop:=st_p182_RightTop.Feedback_2_geat_numerator;
		GearNumeratorGet_LeftBottom:=st_p182_LeftBottom.Feedback_2_geat_numerator;
		GearNumeratorGet_RightBottom:=st_p182_RightBottom.Feedback_2_geat_numerator;
		GearNumeratorGet_PhaseUpper:=st_p182_PhaseUpper.Feedback_2_geat_numerator;
		GearNumeratorGet_PhaseLower:=st_p182_PhaseLower.Feedback_2_geat_numerator;
		//
		GearDenominatorGet_LeftTop:=st_p183_LeftTop.Feedback_2_geat_denominator;
		GearDenominatorGet_RightTop:=st_p183_RightTop.Feedback_2_geat_denominator;
		GearDenominatorGet_LeftBottom:=st_p183_LeftBottom.Feedback_2_geat_denominator;
		GearDenominatorGet_RightBottom:=st_p183_RightBottom.Feedback_2_geat_denominator;
		GearDenominatorGet_PhaseUpper:=st_p183_PhaseUpper.Feedback_2_geat_denominator;
		GearDenominatorGet_PhaseLower:=st_p183_PhaseLower.Feedback_2_geat_denominator;
		//
		Feedback2directionGet_LeftTop:=st_p180_LeftTop.Feedback_direction;
		Feedback2directionGet_RightTop:=st_p180_RightTop.Feedback_direction;
		Feedback2directionGet_LeftBottom:=st_p180_LeftBottom.Feedback_direction;
		Feedback2directionGet_RightBottom:=st_p180_RightBottom.Feedback_direction;
		Feedback2directionGet_PhaseUpper:=st_p180_PhaseUpper.Feedback_direction;
		Feedback2directionGet_PhaseLower:=st_p180_PhaseLower.Feedback_direction;
		//
		IF 	NOT fb_SoEReadDiagMessage_LeftTop.bBusy
			AND NOT fb_SoEReadDiagMessage_RightTop.bBusy
			AND NOT fb_SoEReadDiagMessage_LeftBottom.bBusy
			AND NOT fb_SoEReadDiagMessage_RightBottom.bBusy 
			AND NOT fb_SoEReadDiagMessage_PhaseUpper.bBusy
			AND NOT fb_SoEReadDiagMessage_PhaseLower.bBusy 
			AND NOT FB_SoEReadDiagNumber_LeftTop.bBusy
			AND NOT FB_SoEReadDiagNumber_RightTop.bBusy
			AND NOT FB_SoEReadDiagNumber_LeftBottom.bBusy
			AND NOT FB_SoEReadDiagNumber_RightBottom.bBusy 
			AND NOT FB_SoEReadDiagNumber_PhaseUpper.bBusy
			AND NOT FB_SoEReadDiagNumber_PhaseLower.bBusy 
			AND NOT FB_SoERead_GearNumerator_LeftTop.bBusy 
			AND NOT FB_SoERead_GearNumerator_RightTop.bBusy 
			AND NOT FB_SoERead_GearNumerator_LeftBottom.bBusy 
			AND NOT FB_SoERead_GearNumerator_RightBottom.bBusy 
			AND NOT FB_SoERead_GearNumerator_PhaseUpper.bBusy 
			AND NOT FB_SoERead_GearNumerator_PhaseLower.bBusy 
			AND NOT FB_SoERead_GearDenominator_LeftTop.bBusy 
			AND NOT FB_SoERead_GearDenominator_RightTop.bBusy 
			AND NOT FB_SoERead_GearDenominator_LeftBottom.bBusy 
			AND NOT FB_SoERead_GearDenominator_RightBottom.bBusy 
			AND NOT FB_SoERead_GearDenominator_PhaseUpper.bBusy 
			AND NOT FB_SoERead_GearDenominator_PhaseLower.bBusy 
			AND NOT FB_SoERead_Feedback2direction_LeftTop.bBusy 
			AND NOT FB_SoERead_Feedback2direction_RightTop.bBusy  
			AND NOT FB_SoERead_Feedback2direction_LeftBottom.bBusy 
			AND NOT FB_SoERead_Feedback2direction_RightBottom.bBusy
			AND NOT FB_SoERead_Feedback2direction_PhaseUpper.bBusy 
			AND NOT FB_SoERead_Feedback2direction_PhaseLower.bBusy	THEN
				GetDriveStatusTON2.IN:=TRUE;
				IF GetDriveStatusTON2.Q THEN
					m_GetDriveStatusState:=88;
				END_IF
		END_IF
		IF 	fb_SoEReadDiagMessage_LeftTop.bError
			OR fb_SoEReadDiagMessage_RightTop.bError
			OR fb_SoEReadDiagMessage_LeftBottom.bError
			OR fb_SoEReadDiagMessage_RightBottom.bError
			OR fb_SoEReadDiagMessage_PhaseUpper.bError
			OR fb_SoEReadDiagMessage_PhaseLower.bError
			OR FB_SoEReadDiagNumber_LeftTop.bError
			OR FB_SoEReadDiagNumber_RightTop.bError
			OR FB_SoEReadDiagNumber_LeftBottom.bError
			OR FB_SoEReadDiagNumber_RightBottom.bError 
			OR FB_SoEReadDiagNumber_PhaseUpper.bError
			OR FB_SoEReadDiagNumber_PhaseLower.bError 
			OR FB_SoERead_GearNumerator_LeftTop.bError 
			OR FB_SoERead_GearNumerator_RightTop.bError 
			OR FB_SoERead_GearNumerator_LeftBottom.bError 
			OR FB_SoERead_GearNumerator_RightBottom.bError 
			OR FB_SoERead_GearNumerator_PhaseUpper.bError 
			OR FB_SoERead_GearNumerator_PhaseLower.bError 
			OR FB_SoERead_GearDenominator_LeftTop.bError 
			OR FB_SoERead_GearDenominator_RightTop.bError 
			OR FB_SoERead_GearDenominator_LeftBottom.bError 
			OR FB_SoERead_GearDenominator_RightBottom.bError 
			OR FB_SoERead_GearDenominator_PhaseUpper.bError 
			OR FB_SoERead_GearDenominator_PhaseLower.bError 
			OR FB_SoERead_Feedback2direction_LeftTop.bError 
			OR FB_SoERead_Feedback2direction_RightTop.bError 
			OR FB_SoERead_Feedback2direction_LeftBottom.bError 
			OR FB_SoERead_Feedback2direction_RightBottom.bError 
			OR FB_SoERead_Feedback2direction_PhaseUpper.bError 
			OR FB_SoERead_Feedback2direction_PhaseLower.bError 
		THEN
			m_GetDriveStatusState:=-100;
		END_IF
		
	88:
		bDriveDiagMessageAndNumber:=FALSE;
		A_GetDriverStatusMC();
		GetDriveStatusStateDone:=TRUE;
		GetDriveStatusStateError:=FALSE;
		//
		(*Drive Status*)
		//D012, Axis state machine: Control and power section ready,53266
		IF DriveDiagNumber_LeftTop=16#D012 AND DriveDiagNumber_RightTop=16#D012			
			AND DriveDiagNumber_LeftBottom=16#D012 AND DriveDiagNumber_RightBottom=16#D012
			AND DriveDiagNumber_PhaseUpper=16#D012 AND DriveDiagNumber_PhaseLower=16#D012 THEN
			DriveStatus:=1;
		//D013, Axis state machine: Axis in operation,53267
		ELSIF DriveDiagNumber_LeftTop=16#D013 AND DriveDiagNumber_RightTop=16#D013
			AND DriveDiagNumber_LeftBottom=16#D013 AND DriveDiagNumber_RightBottom=16#D013
			AND DriveDiagNumber_PhaseUpper=16#D013 AND DriveDiagNumber_PhaseLower=16#D013 THEN
			DriveStatus:=2;
		//D014，Axis state machine: Axis halt.53266和53267中间会经历这么一个状态，算正常状态
		ELSIF DriveDiagNumber_LeftTop=16#D014 AND DriveDiagNumber_RightTop=16#D014
			AND DriveDiagNumber_LeftBottom=16#D014 AND DriveDiagNumber_RightBottom=16#D014
			AND DriveDiagNumber_PhaseUpper=16#D014 AND DriveDiagNumber_PhaseLower=16#D014 THEN
			DriveStatus:=3;
		ELSE
			DriveStatus:=0;
		END_IF
		//
		//
		//	//check statusGet and status configured
		IF 	GearNumeratorGet_LeftTop<>GearNumeratorConfigured_LeftTop 
			OR GearNumeratorGet_RightTop<>GearNumeratorConfigured_RightTop
			OR GearNumeratorGet_LeftBottom<>GearNumeratorConfigured_LeftBottom 
			OR GearNumeratorGet_RightBottom<>GearNumeratorConfigured_RightBottom
			OR GearNumeratorGet_PhaseUpper<>GearNumeratorConfigured_PhaseUpper 
			OR GearNumeratorGet_PhaseLower<>GearNumeratorConfigured_PhaseLower
			OR GearDenominatorGet_LeftTop<>GearDenominatorConfigured_LeftTop 
			OR GearDenominatorGet_RightTop<>GearDenominatorConfigured_RightTop
			OR GearDenominatorGet_LeftBottom<>GearDenominatorConfigured_LeftBottom 
			OR GearDenominatorGet_RightBottom<>GearDenominatorConfigured_RightBottom
			OR GearDenominatorGet_PhaseUpper<>GearDenominatorConfigured_PhaseUpper 
			OR GearDenominatorGet_PhaseLower<>GearDenominatorConfigured_PhaseLower THEN
				bDriveDiagMessageAndNumber:=FALSE;
				A_GetDriverStatusMC();
				GetDriveStatusStateDone:=FALSE;
				GetDriveStatusStateError:=TRUE;
				Error:=TRUE;
				ErrorId:=1302;
				ErrorDescription:='gearParameters Error';
				Plc_EmergencyStop:=FALSE;
		END_IF
		IF USELinearEncoder THEN
			IF 	Feedback2directionGet_LeftTop<>Feedback2directionConfigured_LeftTop 
				OR Feedback2directionGet_RightTop<>Feedback2directionConfigured_RightTop
				OR Feedback2directionGet_LeftBottom<>Feedback2directionConfigured_LeftBottom 
				OR Feedback2directionGet_RightBottom<Feedback2directionConfigured_RightBottom 
				OR Feedback2directionGet_PhaseUpper<>Feedback2directionConfigured_PhaseUpper 
				OR Feedback2directionGet_PhaseLower<Feedback2directionConfigured_PhaseLower THEN
					bDriveDiagMessageAndNumber:=FALSE;
					A_GetDriverStatusMC();
					GetDriveStatusStateDone:=FALSE;
					GetDriveStatusStateError:=TRUE;
					Error:=TRUE;
					ErrorId:=1303;
					ErrorDescription:='fb2direction Error';
					Plc_EmergencyStop:=FALSE;
			END_IF 
		END_IF
		m_GetDriveStatusState:=0;
	-100:
		bDriveDiagMessageAndNumber:=FALSE;
		A_GetDriverStatusMC();
		GetDriveStatusStateDone:=FALSE;
		GetDriveStatusStateError:=TRUE;
		Error:=TRUE;
		ErrorId:=1301;
		ErrorDescription:='GetDriveStatusStateError';
END_CASE
END_ACTION

ACTION A_GetDriverStatusMC:
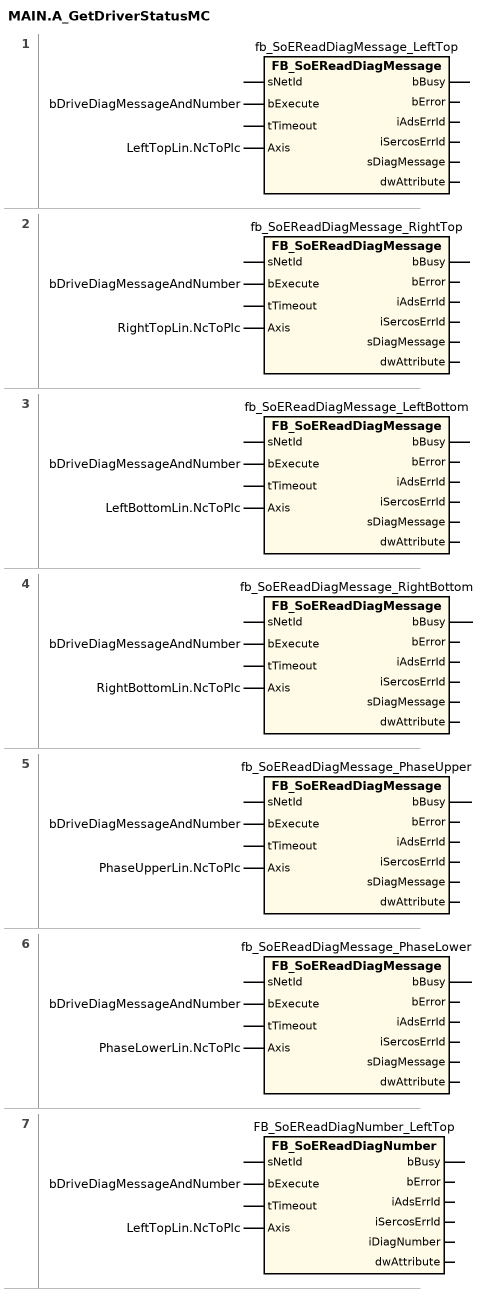
// NETWORK 1
fb_SoEReadDiagMessage_LeftTop(bExecute := bDriveDiagMessageAndNumber, Axis := LeftTopLin.NcToPlc); // FB_SoEReadDiagMessage

// NETWORK 2
fb_SoEReadDiagMessage_RightTop(bExecute := bDriveDiagMessageAndNumber, Axis := RightTopLin.NcToPlc); // FB_SoEReadDiagMessage

// NETWORK 3
fb_SoEReadDiagMessage_LeftBottom(bExecute := bDriveDiagMessageAndNumber, Axis := LeftBottomLin.NcToPlc); // FB_SoEReadDiagMessage

// NETWORK 4
fb_SoEReadDiagMessage_RightBottom(bExecute := bDriveDiagMessageAndNumber, Axis := RightBottomLin.NcToPlc); // FB_SoEReadDiagMessage

// NETWORK 5
fb_SoEReadDiagMessage_PhaseUpper(bExecute := bDriveDiagMessageAndNumber, Axis := PhaseUpperLin.NcToPlc); // FB_SoEReadDiagMessage

// NETWORK 6
fb_SoEReadDiagMessage_PhaseLower(bExecute := bDriveDiagMessageAndNumber, Axis := PhaseLowerLin.NcToPlc); // FB_SoEReadDiagMessage

// NETWORK 7
FB_SoEReadDiagNumber_LeftTop(bExecute := bDriveDiagMessageAndNumber, Axis := LeftTopLin.NcToPlc); // FB_SoEReadDiagNumber

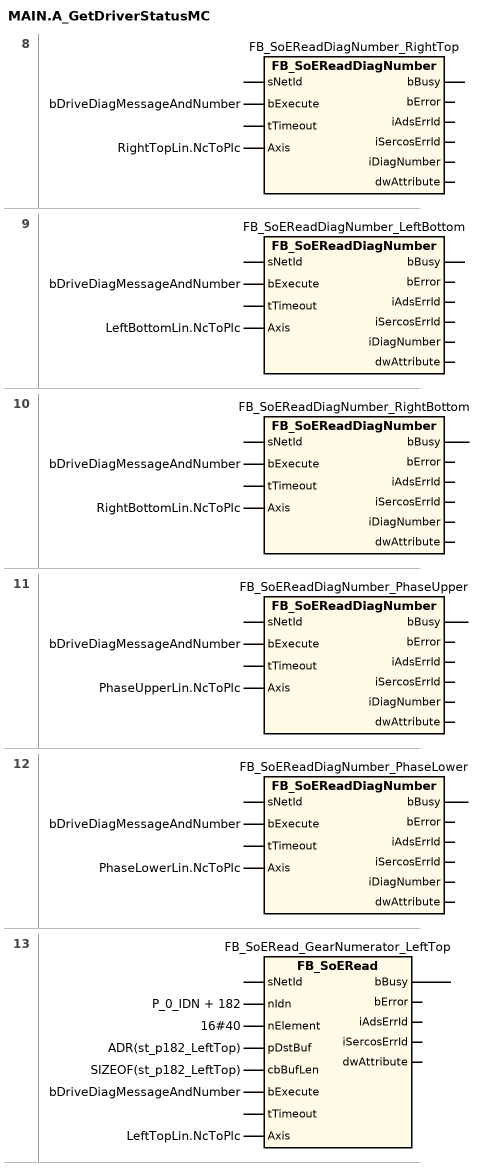
// NETWORK 8
FB_SoEReadDiagNumber_RightTop(bExecute := bDriveDiagMessageAndNumber, Axis := RightTopLin.NcToPlc); // FB_SoEReadDiagNumber

// NETWORK 9
FB_SoEReadDiagNumber_LeftBottom(bExecute := bDriveDiagMessageAndNumber, Axis := LeftBottomLin.NcToPlc); // FB_SoEReadDiagNumber

// NETWORK 10
FB_SoEReadDiagNumber_RightBottom(bExecute := bDriveDiagMessageAndNumber, Axis := RightBottomLin.NcToPlc); // FB_SoEReadDiagNumber

// NETWORK 11
FB_SoEReadDiagNumber_PhaseUpper(bExecute := bDriveDiagMessageAndNumber, Axis := PhaseUpperLin.NcToPlc); // FB_SoEReadDiagNumber

// NETWORK 12
FB_SoEReadDiagNumber_PhaseLower(bExecute := bDriveDiagMessageAndNumber, Axis := PhaseLowerLin.NcToPlc); // FB_SoEReadDiagNumber

// NETWORK 13
FB_SoERead_GearNumerator_LeftTop(
    nIdn := P_0_IDN + 182,
    nElement := 16#40,
    pDstBuf := ADR(st_p182_LeftTop),
    cbBufLen := SIZEOF(st_p182_LeftTop),
    bExecute := bDriveDiagMessageAndNumber,
    Axis := LeftTopLin.NcToPlc); // FB_SoERead

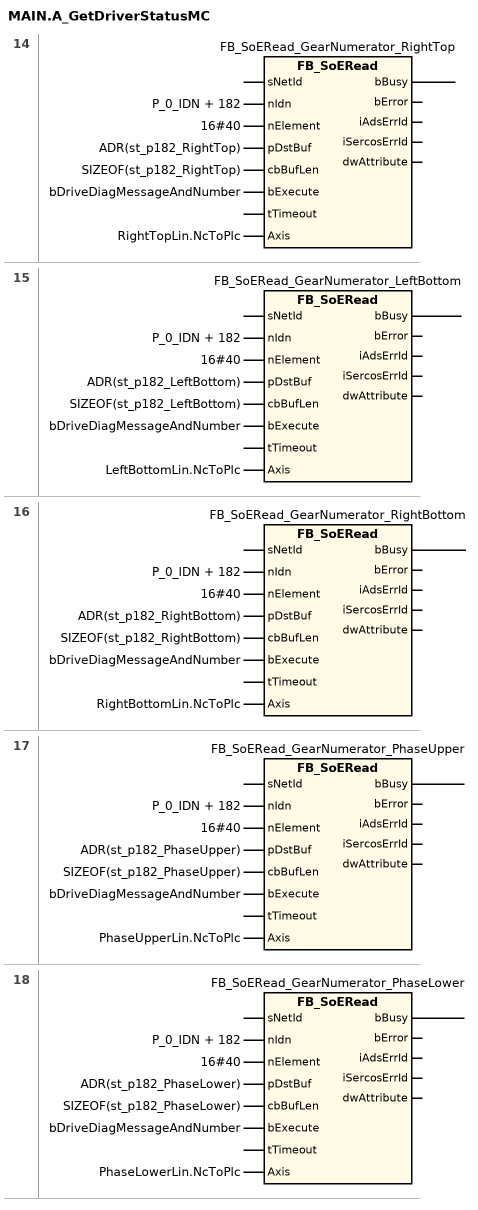
// NETWORK 14
FB_SoERead_GearNumerator_RightTop(
    nIdn := P_0_IDN + 182,
    nElement := 16#40,
    pDstBuf := ADR(st_p182_RightTop),
    cbBufLen := SIZEOF(st_p182_RightTop),
    bExecute := bDriveDiagMessageAndNumber,
    Axis := RightTopLin.NcToPlc); // FB_SoERead

// NETWORK 15
FB_SoERead_GearNumerator_LeftBottom(
    nIdn := P_0_IDN + 182,
    nElement := 16#40,
    pDstBuf := ADR(st_p182_LeftBottom),
    cbBufLen := SIZEOF(st_p182_LeftBottom),
    bExecute := bDriveDiagMessageAndNumber,
    Axis := LeftBottomLin.NcToPlc); // FB_SoERead

// NETWORK 16
FB_SoERead_GearNumerator_RightBottom(
    nIdn := P_0_IDN + 182,
    nElement := 16#40,
    pDstBuf := ADR(st_p182_RightBottom),
    cbBufLen := SIZEOF(st_p182_RightBottom),
    bExecute := bDriveDiagMessageAndNumber,
    Axis := RightBottomLin.NcToPlc); // FB_SoERead

// NETWORK 17
FB_SoERead_GearNumerator_PhaseUpper(
    nIdn := P_0_IDN + 182,
    nElement := 16#40,
    pDstBuf := ADR(st_p182_PhaseUpper),
    cbBufLen := SIZEOF(st_p182_PhaseUpper),
    bExecute := bDriveDiagMessageAndNumber,
    Axis := PhaseUpperLin.NcToPlc); // FB_SoERead

// NETWORK 18
FB_SoERead_GearNumerator_PhaseLower(
    nIdn := P_0_IDN + 182,
    nElement := 16#40,
    pDstBuf := ADR(st_p182_PhaseLower),
    cbBufLen := SIZEOF(st_p182_PhaseLower),
    bExecute := bDriveDiagMessageAndNumber,
    Axis := PhaseLowerLin.NcToPlc); // FB_SoERead

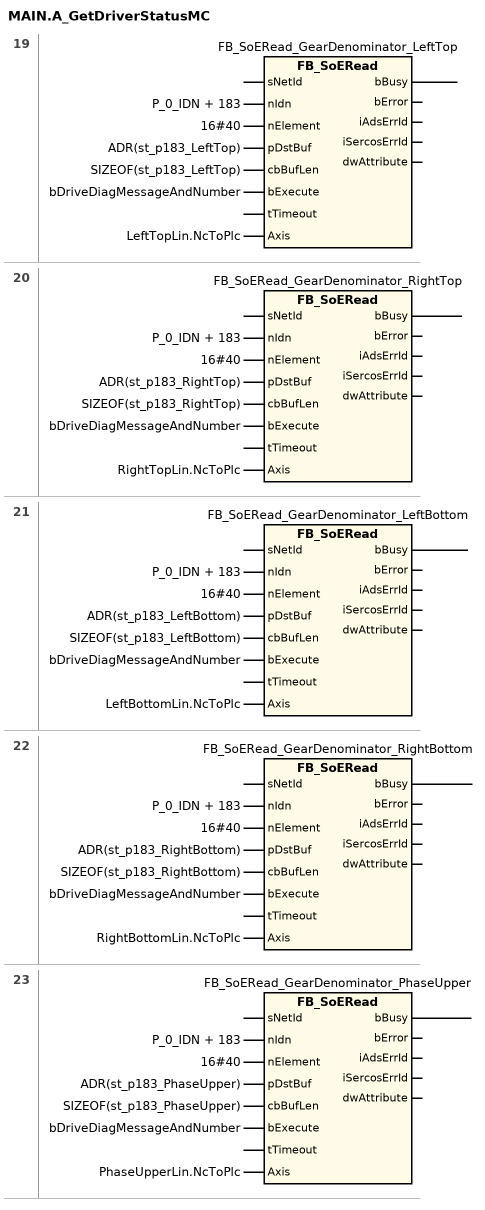
// NETWORK 19
FB_SoERead_GearDenominator_LeftTop(
    nIdn := P_0_IDN + 183,
    nElement := 16#40,
    pDstBuf := ADR(st_p183_LeftTop),
    cbBufLen := SIZEOF(st_p183_LeftTop),
    bExecute := bDriveDiagMessageAndNumber,
    Axis := LeftTopLin.NcToPlc); // FB_SoERead

// NETWORK 20
FB_SoERead_GearDenominator_RightTop(
    nIdn := P_0_IDN + 183,
    nElement := 16#40,
    pDstBuf := ADR(st_p183_RightTop),
    cbBufLen := SIZEOF(st_p183_RightTop),
    bExecute := bDriveDiagMessageAndNumber,
    Axis := RightTopLin.NcToPlc); // FB_SoERead

// NETWORK 21
FB_SoERead_GearDenominator_LeftBottom(
    nIdn := P_0_IDN + 183,
    nElement := 16#40,
    pDstBuf := ADR(st_p183_LeftBottom),
    cbBufLen := SIZEOF(st_p183_LeftBottom),
    bExecute := bDriveDiagMessageAndNumber,
    Axis := LeftBottomLin.NcToPlc); // FB_SoERead

// NETWORK 22
FB_SoERead_GearDenominator_RightBottom(
    nIdn := P_0_IDN + 183,
    nElement := 16#40,
    pDstBuf := ADR(st_p183_RightBottom),
    cbBufLen := SIZEOF(st_p183_RightBottom),
    bExecute := bDriveDiagMessageAndNumber,
    Axis := RightBottomLin.NcToPlc); // FB_SoERead

// NETWORK 23
FB_SoERead_GearDenominator_PhaseUpper(
    nIdn := P_0_IDN + 183,
    nElement := 16#40,
    pDstBuf := ADR(st_p183_PhaseUpper),
    cbBufLen := SIZEOF(st_p183_PhaseUpper),
    bExecute := bDriveDiagMessageAndNumber,
    Axis := PhaseUpperLin.NcToPlc); // FB_SoERead

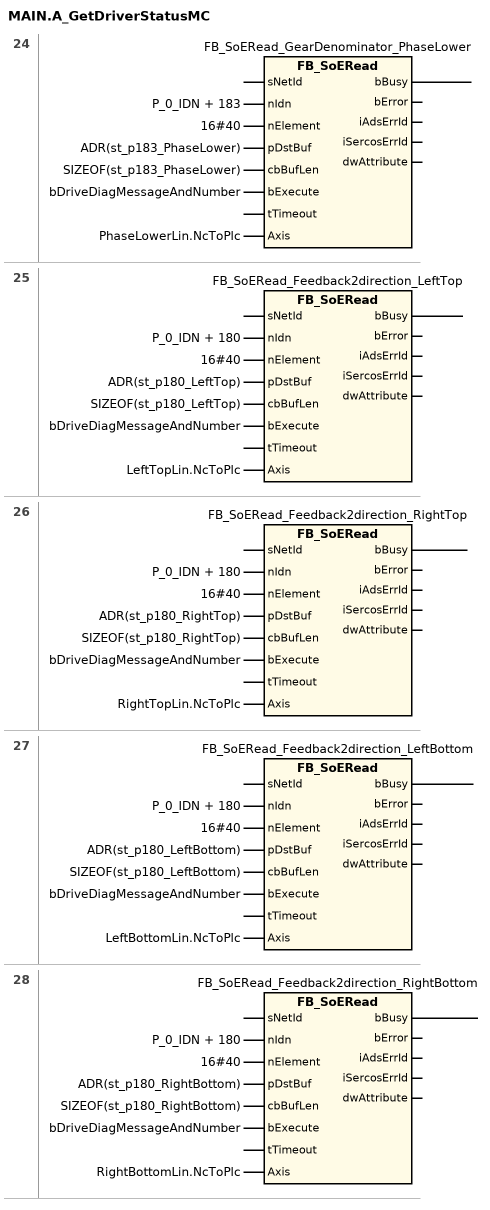
// NETWORK 24
FB_SoERead_GearDenominator_PhaseLower(
    nIdn := P_0_IDN + 183,
    nElement := 16#40,
    pDstBuf := ADR(st_p183_PhaseLower),
    cbBufLen := SIZEOF(st_p183_PhaseLower),
    bExecute := bDriveDiagMessageAndNumber,
    Axis := PhaseLowerLin.NcToPlc); // FB_SoERead

// NETWORK 25
FB_SoERead_Feedback2direction_LeftTop(
    nIdn := P_0_IDN + 180,
    nElement := 16#40,
    pDstBuf := ADR(st_p180_LeftTop),
    cbBufLen := SIZEOF(st_p180_LeftTop),
    bExecute := bDriveDiagMessageAndNumber,
    Axis := LeftTopLin.NcToPlc); // FB_SoERead

// NETWORK 26
FB_SoERead_Feedback2direction_RightTop(
    nIdn := P_0_IDN + 180,
    nElement := 16#40,
    pDstBuf := ADR(st_p180_RightTop),
    cbBufLen := SIZEOF(st_p180_RightTop),
    bExecute := bDriveDiagMessageAndNumber,
    Axis := RightTopLin.NcToPlc); // FB_SoERead

// NETWORK 27
FB_SoERead_Feedback2direction_LeftBottom(
    nIdn := P_0_IDN + 180,
    nElement := 16#40,
    pDstBuf := ADR(st_p180_LeftBottom),
    cbBufLen := SIZEOF(st_p180_LeftBottom),
    bExecute := bDriveDiagMessageAndNumber,
    Axis := LeftBottomLin.NcToPlc); // FB_SoERead

// NETWORK 28
FB_SoERead_Feedback2direction_RightBottom(
    nIdn := P_0_IDN + 180,
    nElement := 16#40,
    pDstBuf := ADR(st_p180_RightBottom),
    cbBufLen := SIZEOF(st_p180_RightBottom),
    bExecute := bDriveDiagMessageAndNumber,
    Axis := RightBottomLin.NcToPlc); // FB_SoERead

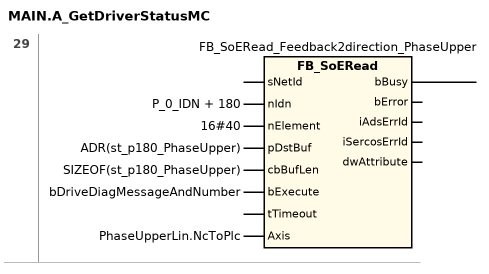
// NETWORK 29
FB_SoERead_Feedback2direction_PhaseUpper(
    nIdn := P_0_IDN + 180,
    nElement := 16#40,
    pDstBuf := ADR(st_p180_PhaseUpper),
    cbBufLen := SIZEOF(st_p180_PhaseUpper),
    bExecute := bDriveDiagMessageAndNumber,
    Axis := PhaseUpperLin.NcToPlc); // FB_SoERead
END_ACTION

ACTION A_GetMotorTemperature:
MotorTemperature_LeftTop:=UINT_TO_LREAL(MotorTemperature[0])/10;
MotorTemperature_RightTop:=UINT_TO_LREAL(MotorTemperature[1])/10;
MotorTemperature_LeftBottom:=UINT_TO_LREAL(MotorTemperature[2])/10;
MotorTemperature_RightBottom:=UINT_TO_LREAL(MotorTemperature[3])/10;
MotorTemperature_PhaseUpper:=UINT_TO_LREAL(MotorTemperature[4])/10;
MotorTemperature_PhaseLower:=UINT_TO_LREAL(MotorTemperature[5])/10;
END_ACTION

ACTION A_GetTemperatureSensorsData:
//sensor_1
dut_sensor_datas_1.data_byte[3]:=Sensor_Reading_1[0];
dut_sensor_datas_1.data_byte[2]:=Sensor_Reading_1[1];
dut_sensor_datas_1.data_byte[1]:=Sensor_Reading_1[2];
dut_sensor_datas_1.data_byte[0]:=Sensor_Reading_1[3];
TemperatureSensors_1:=DINT_TO_LREAL(LREAL_TO_DINT(dut_sensor_datas_1.data_lreal*100))/100;
//sensor_2
dut_sensor_datas_2.data_byte[3]:=Sensor_Reading_2[0];
dut_sensor_datas_2.data_byte[2]:=Sensor_Reading_2[1];
dut_sensor_datas_2.data_byte[1]:=Sensor_Reading_2[2];
dut_sensor_datas_2.data_byte[0]:=Sensor_Reading_2[3];
TemperatureSensors_2:=DINT_TO_LREAL(LREAL_TO_DINT(dut_sensor_datas_2.data_lreal*100))/100;
//sensor_3
dut_sensor_datas_3.data_byte[3]:=Sensor_Reading_3[0];
dut_sensor_datas_3.data_byte[2]:=Sensor_Reading_3[1];
dut_sensor_datas_3.data_byte[1]:=Sensor_Reading_3[2];
dut_sensor_datas_3.data_byte[0]:=Sensor_Reading_3[3];
TemperatureSensors_3:=DINT_TO_LREAL(LREAL_TO_DINT(dut_sensor_datas_3.data_lreal*100))/100;
//sensor_4
dut_sensor_datas_4.data_byte[3]:=Sensor_Reading_4[0];
dut_sensor_datas_4.data_byte[2]:=Sensor_Reading_4[1];
dut_sensor_datas_4.data_byte[1]:=Sensor_Reading_4[2];
dut_sensor_datas_4.data_byte[0]:=Sensor_Reading_4[3];
TemperatureSensors_4:=DINT_TO_LREAL(LREAL_TO_DINT(dut_sensor_datas_4.data_lreal*100))/100;
//sensor_5
dut_sensor_datas_5.data_byte[3]:=Sensor_Reading_5[0];
dut_sensor_datas_5.data_byte[2]:=Sensor_Reading_5[1];
dut_sensor_datas_5.data_byte[1]:=Sensor_Reading_5[2];
dut_sensor_datas_5.data_byte[0]:=Sensor_Reading_5[3];
TemperatureSensors_5:=DINT_TO_LREAL(LREAL_TO_DINT(dut_sensor_datas_5.data_lreal*100))/100;
//sensor_6
dut_sensor_datas_6.data_byte[3]:=Sensor_Reading_6[0];
dut_sensor_datas_6.data_byte[2]:=Sensor_Reading_6[1];
dut_sensor_datas_6.data_byte[1]:=Sensor_Reading_6[2];
dut_sensor_datas_6.data_byte[0]:=Sensor_Reading_6[3];
TemperatureSensors_6:=DINT_TO_LREAL(LREAL_TO_DINT(dut_sensor_datas_6.data_lreal*100))/100;
//sensor_7
dut_sensor_datas_7.data_byte[3]:=Sensor_Reading_7[0];
dut_sensor_datas_7.data_byte[2]:=Sensor_Reading_7[1];
dut_sensor_datas_7.data_byte[1]:=Sensor_Reading_7[2];
dut_sensor_datas_7.data_byte[0]:=Sensor_Reading_7[3];
TemperatureSensors_7:=DINT_TO_LREAL(LREAL_TO_DINT(dut_sensor_datas_7.data_lreal*100))/100;
//sensor_8
dut_sensor_datas_8.data_byte[3]:=Sensor_Reading_8[0];
dut_sensor_datas_8.data_byte[2]:=Sensor_Reading_8[1];
dut_sensor_datas_8.data_byte[1]:=Sensor_Reading_8[2];
dut_sensor_datas_8.data_byte[0]:=Sensor_Reading_8[3];
TemperatureSensors_8:=DINT_TO_LREAL(LREAL_TO_DINT(dut_sensor_datas_8.data_lreal*100))/100;
//计算temperature_gradient
temperature_gradient_2_To_1:=ABS(TemperatureSensors_2-TemperatureSensors_1);
temperature_gradient_3_To_2:=ABS(TemperatureSensors_3-TemperatureSensors_2);
temperature_gradient_5_To_4:=ABS(TemperatureSensors_5-TemperatureSensors_4);
temperature_gradient_6_To_5:=ABS(TemperatureSensors_6-TemperatureSensors_5);
temperature_gradient_max:=DINT_TO_LREAL(LREAL_TO_DINT(MAX(temperature_gradient_2_To_1,temperature_gradient_3_To_2,
							temperature_gradient_5_To_4,temperature_gradient_6_To_5)*100))/100;
//计算大梁上的温度平均值
temperature_average:=DINT_TO_LREAL(LREAL_TO_DINT((TemperatureSensors_1+TemperatureSensors_2+TemperatureSensors_3+TemperatureSensors_4
					+TemperatureSensors_5+TemperatureSensors_6)/6*100))/100;
					

//传感器温度状态：0：有传感器度数错误；1:常温；2:低温；3:常温和低温中间态
IF TemperatureSensors_1=0 OR TemperatureSensors_2=0 OR TemperatureSensors_3=0 
	OR TemperatureSensors_4=0 OR TemperatureSensors_5=0 OR TemperatureSensors_6=0 THEN	
	temperatureStatus:=0;//有传感器读数错误
ELSIF TemperatureSensors_1>=RoomTemperatureThreshold AND TemperatureSensors_2>=RoomTemperatureThreshold AND TemperatureSensors_3>=RoomTemperatureThreshold
	AND TemperatureSensors_4>=RoomTemperatureThreshold AND TemperatureSensors_5>=RoomTemperatureThreshold AND TemperatureSensors_6>=RoomTemperatureThreshold THEN	
	temperatureStatus:=1;//常温
ELSIF TemperatureSensors_1<=CryogenicTemperatureThreshold AND TemperatureSensors_1>77
	AND TemperatureSensors_2<=CryogenicTemperatureThreshold  AND TemperatureSensors_2>77
	AND TemperatureSensors_3<=CryogenicTemperatureThreshold  AND TemperatureSensors_3>77
	AND TemperatureSensors_4<=CryogenicTemperatureThreshold   AND TemperatureSensors_4>77
	AND TemperatureSensors_5<=CryogenicTemperatureThreshold  AND TemperatureSensors_5>77
	AND TemperatureSensors_6<=CryogenicTemperatureThreshold   AND TemperatureSensors_6>77 THEN	
	temperatureStatus:=2;//低温
ELSE
	temperatureStatus:=3;//常温和低温中间
END_IF
END_ACTION

ACTION A_InitAxisParameters:
(*ÖáÎ»ÖÃ¡¢ËÙ¶È¡¢PosDiff*)

	Pos_LeftTopLin:=DINT_TO_LREAL(LREAL_TO_DINT(LeftTopLin.NcToPlc.ActPos*100000))/100000;
	Pos_RightTopLin:=DINT_TO_LREAL(LREAL_TO_DINT(RightTopLin.NcToPlc.ActPos*100000))/100000;
	Pos_LeftBottomLin:=DINT_TO_LREAL(LREAL_TO_DINT(LeftBottomLin.NcToPlc.ActPos*100000))/100000;
	Pos_RightBottomLin:=DINT_TO_LREAL(LREAL_TO_DINT(RightBottomLin.NcToPlc.ActPos*100000))/100000;
	Pos_PhaseUpperLin:=DINT_TO_LREAL(LREAL_TO_DINT(PhaseUpperLin.NcToPlc.ActPos*100000))/100000;
	Pos_PhaseLowerLin:=DINT_TO_LREAL(LREAL_TO_DINT(PhaseLowerLin.NcToPlc.ActPos*100000))/100000;
	
	moveStatusLeftTop:=LeftTopLin.Status.Moving;
	moveStatusRightTop:=RightTopLin.Status.Moving;
	moveStatusLeftBottom:=LeftBottomLin.Status.Moving;
	moveStatusRightBottom:=RightBottomLin.Status.Moving;
	moveStatusPhaseUpper:=PhaseUpperLin.Status.Moving;
	moveStatusPhaseLower:=PhaseLowerLin.Status.Moving;
	
	moveStatusAllAxis:=moveStatusLeftTop AND moveStatusRightTop AND moveStatusLeftBottom AND moveStatusRightBottom;
	moveStatusAnyAxis:=moveStatusLeftTop OR moveStatusRightTop OR moveStatusLeftBottom OR moveStatusRightBottom;	
	Velo_LeftTopLin:=DINT_TO_LREAL(LREAL_TO_DINT(LeftTopLin.NcToPlc.ActVelo*100000))/100000;
	Velo_RightTopLin:=DINT_TO_LREAL(LREAL_TO_DINT(RightTopLin.NcToPlc.ActVelo*100000))/100000;
	Velo_LeftBottomLin:=DINT_TO_LREAL(LREAL_TO_DINT(LeftBottomLin.NcToPlc.ActVelo*100000))/100000;
	Velo_RightBottomLin:=DINT_TO_LREAL(LREAL_TO_DINT(RightBottomLin.NcToPlc.ActVelo*100000))/100000;
	Velo_PhaseUpperLin:=DINT_TO_LREAL(LREAL_TO_DINT(PhaseUpperLin.NcToPlc.ActVelo*100000))/100000;
	Velo_PhaseLowerLin:=DINT_TO_LREAL(LREAL_TO_DINT(PhaseLowerLin.NcToPlc.ActVelo*100000))/100000;
	
	PosDiff_LeftTopLin_actual:=DINT_TO_LREAL(LREAL_TO_DINT(LeftTopLin.NcToPlc.PosDiff*100000))/100000;
	PosDiff_RightTopLin_actual:=DINT_TO_LREAL(LREAL_TO_DINT(RightTopLin.NcToPlc.PosDiff*100000))/100000;
	PosDiff_LeftBottomLin_actual:=DINT_TO_LREAL(LREAL_TO_DINT(LeftBottomLin.NcToPlc.PosDiff*100000))/100000;
	PosDiff_RightBottomLin_actual:=DINT_TO_LREAL(LREAL_TO_DINT(RightBottomLin.NcToPlc.PosDiff*100000))/100000;
	PosDiff_PhaseUpperLin_actual:=DINT_TO_LREAL(LREAL_TO_DINT(PhaseUpperLin.NcToPlc.PosDiff*100000))/100000;
	PosDiff_PhaseLowerLin_actual:=DINT_TO_LREAL(LREAL_TO_DINT(PhaseLowerLin.NcToPlc.PosDiff*100000))/100000;;

	//Torque
	Torque_LeftTopLin:=LeftTopLin.NcToPlc.ActTorque;
	Torque_RightTopLin:=RightTopLin.NcToPlc.ActTorque;
	Torque_LeftBottomLin:=LeftBottomLin.NcToPlc.ActTorque;
	Torque_RightBottomLin:=RightBottomLin.NcToPlc.ActTorque;
	Torque_PhaseUpperLin:=LeftBottomLin.NcToPlc.ActTorque;
	Torque_PhaseLowerLin:=RightBottomLin.NcToPlc.ActTorque;
	
	LeftTopLin.ReadStatus();
	RightTopLin.ReadStatus();
	LeftBottomLin.ReadStatus();
	RightBottomLin.ReadStatus();
	PhaseUpperLin.ReadStatus();
	PhaseLowerLin.ReadStatus();

(*Motor Pos Velo Lagdistance status get*)
	//Position
	Pos_LeftTopMotor:=DINT_TO_LREAL(LREAL_TO_DINT(LeftTopMotor.NcToPlc.ActPos*100000))/100000;
	Pos_RightTopMotor:=DINT_TO_LREAL(LREAL_TO_DINT(RightTopMotor.NcToPlc.ActPos*100000))/100000;
	Pos_LeftBottomMotor:=DINT_TO_LREAL(LREAL_TO_DINT(LeftBottomMotor.NcToPlc.ActPos*100000))/100000;
	Pos_RightBottomMotor:=DINT_TO_LREAL(LREAL_TO_DINT(RightBottomMotor.NcToPlc.ActPos*100000))/100000;
	Pos_PhaseUpperMotor:=DINT_TO_LREAL(LREAL_TO_DINT(PhaseUpperMotor.NcToPlc.ActPos*100000))/100000;
	Pos_PhaseLowerMotor:=DINT_TO_LREAL(LREAL_TO_DINT(PhaseLowerMotor.NcToPlc.ActPos*100000))/100000;
	//Moving status
	moveStatusLeftTopMotor:=LeftTopMotor.Status.Moving;
	moveStatusRightTopMotor:=RightTopMotor.Status.Moving;
	moveStatusLeftBottomMotor:=LeftBottomMotor.Status.Moving;
	moveStatusRightBottomMotor:=RightBottomMotor.Status.Moving;
	moveStatusPhaseUpperMotor:=PhaseUpperMotor.Status.Moving;
	moveStatusPhaseLowerMotor:=PhaseLowerMotor.Status.Moving;
	moveStatusAllAxisMotor:=moveStatusLeftTopMotor AND moveStatusRightTopMotor AND moveStatusLeftBottomMotor AND moveStatusRightBottomMotor;
	moveStatusAnyAxisMotor:=moveStatusLeftTopMotor OR moveStatusRightTopMotor OR moveStatusLeftBottomMotor OR moveStatusRightBottomMotor;
	//Velocity
	Velo_LeftTopMotor:=DINT_TO_LREAL(LREAL_TO_DINT(LeftTopMotor.NcToPlc.ActVelo*100000))/100000;
	Velo_RightTopMotor:=DINT_TO_LREAL(LREAL_TO_DINT(RightTopMotor.NcToPlc.ActVelo*100000))/100000;
	Velo_LeftBottomMotor:=DINT_TO_LREAL(LREAL_TO_DINT(LeftBottomMotor.NcToPlc.ActVelo*100000))/100000;
	Velo_RightBottomMotor:=DINT_TO_LREAL(LREAL_TO_DINT(RightBottomMotor.NcToPlc.ActVelo*100000))/100000;
	Velo_PhaseUpperMotor:=DINT_TO_LREAL(LREAL_TO_DINT(PhaseUpperMotor.NcToPlc.ActVelo*100000))/100000;
	Velo_PhaseLowerMotor:=DINT_TO_LREAL(LREAL_TO_DINT(PhaseLowerMotor.NcToPlc.ActVelo*100000))/100000;
	//LagDistance
	PosDiff_LeftTopMotor_actual:=DINT_TO_LREAL(LREAL_TO_DINT(LeftTopMotor.NcToPlc.PosDiff*100000))/100000;
	PosDiff_RightTopMotor_actual:=DINT_TO_LREAL(LREAL_TO_DINT(RightTopMotor.NcToPlc.PosDiff*100000))/100000;
	PosDiff_LeftBottomMotor_actual:=DINT_TO_LREAL(LREAL_TO_DINT(LeftBottomMotor.NcToPlc.PosDiff*100000))/100000;
	PosDiff_RightBottomMotor_actual:=DINT_TO_LREAL(LREAL_TO_DINT(RightBottomMotor.NcToPlc.PosDiff*100000))/100000;
	PosDiff_PhaseUpperMotor_actual:=DINT_TO_LREAL(LREAL_TO_DINT(PhaseUpperMotor.NcToPlc.PosDiff*100000))/100000;
	PosDiff_PhaseLowerMotor_actual:=DINT_TO_LREAL(LREAL_TO_DINT(PhaseLowerMotor.NcToPlc.PosDiff*100000))/100000;
	//Torque
	Torque_LeftTopMotor:=LeftTopMotor.NcToPlc.ActTorque;
	Torque_RightTopMotor:=RightTopMotor.NcToPlc.ActTorque;
	Torque_LeftBottomMotor:=LeftBottomMotor.NcToPlc.ActTorque;
	Torque_RightBottomMotor:=RightBottomMotor.NcToPlc.ActTorque;
	Torque_PhaseUpperMotor:=PhaseUpperMotor.NcToPlc.ActTorque;
	Torque_PhaseLowerMotor:=PhaseLowerMotor.NcToPlc.ActTorque;

	LeftTopMotor.ReadStatus();
	RightTopMotor.ReadStatus();
	LeftBottomMotor.ReadStatus();
	RightBottomMotor.ReadStatus();
	PhaseUpperMotor.ReadStatus();
	PhaseLowerMotor.ReadStatus();
	//
	//get Delta
	//
	//Delta Pos
	DeltaPos_LeftTop:=Pos_LeftTopLin - Pos_LeftTopMotor;
	DeltaPos_RightTop:=Pos_RightTopLin - Pos_RightTopMotor;
	DeltaPos_LeftBottom:=Pos_LeftBottomLin - Pos_LeftBottomMotor;
	DeltaPos_RightBottom:=Pos_RightBottomLin - Pos_RightBottomMotor;
	DeltaPos_PhaseUpper:=Pos_PhaseUpperLin - Pos_PhaseUpperMotor;
	DeltaPos_PhaseLower:=Pos_PhaseLowerLin - Pos_PhaseLowerMotor;
	//Delta Velocity	
	DeltaVelo_LeftTop:=Velo_LeftTopLin - Velo_LeftTopMotor;
	DeltaVelo_RightTop:=Velo_RightTopLin - Velo_RightTopMotor;
	DeltaVelo_LeftBottom:=Velo_LeftBottomLin - Velo_LeftBottomMotor;
	DeltaVelo_RightBottom:=Velo_RightBottomLin - Velo_RightBottomMotor;
	DeltaVelo_PhaseUpper:=Velo_PhaseUpperLin - Velo_PhaseUpperMotor;
	DeltaVelo_PhaseLower:=Velo_PhaseLowerLin - Velo_PhaseLowerMotor;
	//Delta lagDistance
	DeltaPosDiff_LeftTop_actual:=PosDiff_LeftTopLin_actual - PosDiff_LeftTopMotor_actual;
	DeltaPosDiff_RightTop_actual:=PosDiff_RightTopLin_actual - PosDiff_RightTopMotor_actual;
	DeltaPosDiff_LeftBottom_actual:=PosDiff_LeftBottomLin_actual - PosDiff_LeftBottomMotor_actual;
	DeltaPosDiff_RightBottom_actual:=PosDiff_RightBottomLin_actual - PosDiff_RightBottomMotor_actual;	
	DeltaPosDiff_PhaseUpper_actual:=PosDiff_PhaseUpperLin_actual - PosDiff_PhaseUpperMotor_actual;
	DeltaPosDiff_PhaseLower_actual:=PosDiff_PhaseLowerLin_actual - PosDiff_PhaseLowerMotor_actual;	
	//Delta Torque
	DeltaTorque_LeftTop:=Torque_LeftTopLin - Torque_LeftTopMotor;
	DeltaTorque_RightTop:=Torque_RightTopLin - Torque_RightTopMotor;
	DeltaTorque_LeftBottom:=Torque_LeftBottomLin -Torque_LeftBottomMotor;
	DeltaTorque_RightBottom:=Torque_RightBottomLin - Torque_RightBottomMotor;
	DeltaTorque_PhaseUpper:=Torque_PhaseUpperLin -Torque_PhaseUpperMotor;
	DeltaTorque_PhaseLower:=Torque_PhaseLowerLin - Torque_PhaseLowerMotor;
END_ACTION

ACTION A_InitRecipeParameters:
CASE state_loadParameters OF
	0:
		LoadParameter:=TRUE;
		Read_R_TRIG(CLK:=LoadParameter , Q=> );
		IF Read_R_TRIG.Q THEN
			state_loadParameters:=1;
		END_IF
	1:
		 ReturnDwordLoad:=RecipeManCommands.LoadAndWriteRecipe(RecipeDefinitionName:='Recipes' , RecipeName:='ParametersAK');
    	 LoadParameter:=FALSE;
		 IF ReturnDwordLoad<>0 THEN
		 	state_loadParameters:=-100;
		ELSE
			LoadRecipeParameters:=TRUE;
			LoadParameter:=FALSE;
			state_loadParameters:=88;
	 	END_IF
	88:
		loadParametersDone:=TRUE;
	-100:
		loadParametersDone:=FALSE;
		Error:=TRUE;
		ErrorId:=101;
		ErrorDescription:='LoadRecipeParameters Error';
		Plc_EmergencyStop:=FALSE;
END_CASE

////Save_R_TRIG(CLK:=SaveParameter , Q=> );
//Read_R_TRIG(CLK:=LoadParameter , Q=> );
//IF Save_R_TRIG.Q THEN  //将plc数据以文件形式保存在工控机中
//	 RecipeManCommands.CreateRecipe(RecipeDefinitionName:='Recipes' , RecipeName:='Parameters' );
//	 RecipeManCommands.ReadAndSaveRecipe(RecipeDefinitionName:='Recipes' , RecipeName:='Parameters' );
//	 SaveParameter:=FALSE;
//END_IF
//IF Read_R_TRIG.Q THEN  //将工控机中的文件数据读取到plc中
//     ReturnDwordLoad:=RecipeManCommands.LoadAndWriteRecipe(RecipeDefinitionName:='Recipes' , RecipeName:='Parameters');
//     LoadParameter:=FALSE;
//	 IF ReturnDwordLoad<>0 THEN
//		 Error:=TRUE;
//		 ErrorId:=101;
//		 ErrorDescription:='LoadRecipeParameters Error';
//		 Plc_EmergencyStop:=FALSE;
//	 END_IF
//END_IF
END_ACTION

ACTION A_KillOpcIocShellExe:
R_TRIG_Exekill(CLK:=bExe_Kill_Prog, Q=> );
CASE Exe_kill_step OF
	0:
		IF R_TRIG_Exekill.Q THEN
			NT_StartProcess_Kill.START:=FALSE;
			NT_StartProcess_Kill.PATHSTR:='C:\HZB\OpcIocShell\IDControlIOC\killcmd.bat';
			//NT_StartProcess_Kill.DIRNAME:='C:\Program Files (x86)\HZB\OpcIocShell\bin\opcIocShell.exe';
			Exe_kill_step:=10;
		END_IF;
	10:
		NT_StartProcess_Kill.START:=TRUE;
		Exe_kill_step:=20;
	20:
		IF NT_StartProcess_Kill.ERR THEN
			Exe_kill_step:=0;
		ELSE
			Exe_kill_step:=30;
		END_IF;

	30:
		NT_StartProcess_Kill.START:=TRUE;
		Exe_kill_step:=40;
	40:
		IF NOT NT_StartProcess_Kill.BUSY THEN
			NT_StartProcess_Kill.START:=FALSE;
			Exe_Kill_Done:=TRUE;
			Exe_kill_step:=0;
		END_IF;
END_CASE;

NT_StartProcess_Kill(
	NETID:='' ,
	PATHSTR:= ,
	DIRNAME:= , 
	COMNDLINE:= , 
	START:= ,
	ERRID=> );
END_ACTION

ACTION A_LEHeartBeatMonitor:
//monitor only while power on and not simulation or not use LE
IF NOT st_Power THEN
	RETURN;
END_IF
(**)
IF simulation THEN
	RETURN;
END_IF
IF NOT USELinearEncoder THEN
	RETURN;
END_IF

// 初始化
IF LEHeartBeatFirstScan THEN
    Velo_LeftTopLin_Last := LeftTopLin.NcToPlc.ActVelo;
    Velo_RightTopLin_Last := RightTopLin.NcToPlc.ActVelo;
    Velo_LeftBottomLin_Last := LeftBottomLin.NcToPlc.ActVelo;
    Velo_RightBottomLin_Last := RightBottomLin.NcToPlc.ActVelo;
    Velo_PhaseUpperLin_Last := PhaseUpperLin.NcToPlc.ActVelo;
    Velo_PhaseLowerLin_Last := PhaseLowerLin.NcToPlc.ActVelo;
    LEHeartBeatFirstScan := FALSE;
END_IF;

// 计算光栅前后速度差，速度差比位置差更敏感
DeltaVelo_LeftTopLin := ABS(LeftTopLin.NcToPlc.ActVelo - Velo_LeftTopLin_Last);
DeltaVelo_RightTopLin := ABS(RightTopLin.NcToPlc.ActVelo - Velo_RightTopLin_Last);
DeltaVelo_LeftBottomLin := ABS(LeftBottomLin.NcToPlc.ActVelo - Velo_LeftBottomLin_Last);
DeltaVelo_RightBottomLin := ABS(RightBottomLin.NcToPlc.ActVelo - Velo_RightBottomLin_Last);
DeltaVelo_PhaseUpperLin := ABS(PhaseUpperLin.NcToPlc.ActVelo - Velo_PhaseUpperLin_Last);
DeltaVelo_PhaseLowerLin := ABS(PhaseLowerLin.NcToPlc.ActVelo - Velo_PhaseLowerLin_Last);
//LeftTop monitor
IF DeltaVelo_LeftTopLin > LEHeartBeatDeadZone THEN
    // 有变动，光栅正常，计数器归零，更新位置,重置所有状态
    StableTimer_LeftTopLin(IN := FALSE, PT := LEHeartBeatAlarmTime);
    Alarm_LeftTopLin := FALSE;
    Velo_LeftTopLin_Last := LeftTopLin.NcToPlc.ActVelo;  // 
    StableTime_LeftTopLin := T#0S;
	IsInitialPositionSet_LeftTop:=FALSE;
	Alarm_LeftTopMotorPos:=FALSE;
	Alarm_LeftTopMotorVelo:=FALSE;
ELSE
    //一点变动没有了，光栅异常，开始计时
    StableTimer_LeftTopLin(
        IN := TRUE,
        PT := LEHeartBeatAlarmTime,
        ET => StableTime_LeftTopLin
    );
	//记录电机初始位置，后后续对比做准备
	IF NOT IsInitialPositionSet_LeftTop THEN
        Pos_LeftTopMotor_Initial := Pos_LeftTopMotor;  // 记录初始位置
        IsInitialPositionSet_LeftTop := TRUE;
   	END_IF;
    
    // 100ms速度完全不变，开始监控电机速度和位置
    IF StableTimer_LeftTopLin.Q THEN
        Alarm_LeftTopLin := TRUE;  // 
			//电机位置对比及监测
			MotorPosChange_LeftTop:=ABS( Pos_LeftTopMotor-Pos_LeftTopMotor_Initial);
			IF MotorPosChange_LeftTop > Threshold_LeftTopMotorPos THEN
				Alarm_LeftTopMotorPos:=TRUE;
				ErrorID:=5001;
				ErrorDescription:='5001';
				Error:=TRUE;
				FB_PlcEmergencyStop();
				LED_Error:=TRUE;
			ELSE
				Alarm_LeftTopMotorPos:=FALSE;
			END_IF
			//电机速度监测
			IF Velo_LeftTopMotor > Threshold_LeftTopMotorVelo THEN
				Alarm_LeftTopMotorVelo:=TRUE;
				ErrorID:=5002;
				ErrorDescription:='5002';
				Error:=TRUE;
				FB_PlcEmergencyStop();
				LED_Error:=TRUE;
			ELSE
				Alarm_LeftTopMotorVelo:=FALSE;
			END_IF
    ELSE
        Alarm_LeftTopLin := FALSE;
	END_IF
END_IF
//RightTop monitor
IF DeltaVelo_RightTopLin > LEHeartBeatDeadZone THEN
    // 有变动，光栅正常，计数器归零，更新位置,重置所有状态
    StableTimer_RightTopLin(IN := FALSE, PT := LEHeartBeatAlarmTime);
    Alarm_RightTopLin := FALSE;
    Velo_RightTopLin_Last := RightTopLin.NcToPlc.ActVelo;  // 
    StableTime_RightTopLin := T#0S;
	IsInitialPositionSet_RightTop:=FALSE;
	Alarm_RightTopMotorPos:=FALSE;
	Alarm_RightTopMotorVelo:=FALSE;
ELSE
    //一点变动没有了，光栅异常，开始计时
    StableTimer_RightTopLin(
        IN := TRUE,
        PT :=LEHeartBeatAlarmTime,
        ET => StableTime_RightTopLin
    );
	//记录电机初始位置，后后续对比做准备
	IF NOT IsInitialPositionSet_RightTop THEN
        Pos_RightTopMotor_Initial := Pos_RightTopMotor;  // 记录初始位置
        IsInitialPositionSet_RightTop := TRUE;
   	END_IF;
    
    // 100ms速度完全不变，开始监控电机速度和位置
    IF StableTimer_RightTopLin.Q THEN
        Alarm_RightTopLin := TRUE;  // 
			//电机位置对比及监测
			MotorPosChange_RightTop:=ABS( Pos_RightTopMotor-Pos_RightTopMotor_Initial);
			IF MotorPosChange_RightTop > Threshold_RightTopMotorPos THEN
				Alarm_RightTopMotorPos:=TRUE;
				ErrorID:=5003;
				ErrorDescription:='5003';
				Error:=TRUE;
				FB_PlcEmergencyStop();
				LED_Error:=TRUE;
			ELSE
				Alarm_RightTopMotorPos:=FALSE;
			END_IF
			//电机速度监测
			IF Velo_RightTopMotor > Threshold_RightTopMotorVelo THEN
				Alarm_RightTopMotorVelo:=TRUE;
				ErrorID:=5004;
				ErrorDescription:='5004';
				Error:=TRUE;
				FB_PlcEmergencyStop();
				LED_Error:=TRUE;
			ELSE
				Alarm_RightTopMotorVelo:=FALSE;
			END_IF
    ELSE
        Alarm_RightTopLin := FALSE;
	END_IF
END_IF
//LeftBottom monitor
IF DeltaVelo_LeftBottomLin > LEHeartBeatDeadZone THEN
    // 有变动，光栅正常，计数器归零，更新位置,重置所有状态
    StableTimer_LeftBottomLin(IN := FALSE, PT := LEHeartBeatAlarmTime);
    Alarm_LeftBottomLin := FALSE;
    Velo_LeftBottomLin_Last := LeftBottomLin.NcToPlc.ActVelo;  // 
    StableTime_LeftBottomLin := T#0S;
	IsInitialPositionSet_LeftBottom:=FALSE;
	Alarm_LeftBottomMotorPos:=FALSE;
	Alarm_LeftBottomMotorVelo:=FALSE;
ELSE
    //一点变动没有了，光栅异常，开始计时
    StableTimer_LeftBottomLin(
        IN := TRUE,
        PT := LEHeartBeatAlarmTime,
        ET => StableTime_LeftBottomLin
    );
	//记录电机初始位置，后后续对比做准备
	IF NOT IsInitialPositionSet_LeftBottom THEN
        Pos_LeftBottomMotor_Initial := Pos_LeftBottomMotor;  // 记录初始位置
        IsInitialPositionSet_LeftBottom := TRUE;
   	END_IF;
    
    // 100ms速度完全不变，开始监控电机速度和位置
    IF StableTimer_LeftBottomLin.Q THEN
        Alarm_LeftBottomLin := TRUE;  // 
			//电机位置对比及监测
			MotorPosChange_LeftBottom:=ABS( Pos_LeftBottomMotor-Pos_LeftBottomMotor_Initial);
			IF MotorPosChange_LeftBottom > Threshold_LeftBottomMotorPos THEN
				Alarm_LeftBottomMotorPos:=TRUE;
				ErrorID:=5005;
				ErrorDescription:='5005';
				Error:=TRUE;
				FB_PlcEmergencyStop();
				LED_Error:=TRUE;
			ELSE
				Alarm_LeftBottomMotorPos:=FALSE;
			END_IF
			//电机速度监测
			IF Velo_LeftBottomMotor > Threshold_LeftBottomMotorVelo THEN
				Alarm_LeftBottomMotorVelo:=TRUE;
				ErrorID:=5006;
				ErrorDescription:='5006';
				Error:=TRUE;
				FB_PlcEmergencyStop();
				LED_Error:=TRUE;
			ELSE
				Alarm_LeftBottomMotorVelo:=FALSE;
			END_IF
    ELSE
        Alarm_LeftBottomLin := FALSE;
	END_IF
END_IF
//RightBottom monitor
IF DeltaVelo_RightBottomLin > LEHeartBeatDeadZone THEN
    // 有变动，光栅正常，计数器归零，更新位置,重置所有状态
    StableTimer_RightBottomLin(IN := FALSE, PT := LEHeartBeatAlarmTime);
    Alarm_RightBottomLin := FALSE;
    Velo_RightBottomLin_Last := RightBottomLin.NcToPlc.ActVelo;  // 
    StableTime_RightBottomLin := T#0S;
	IsInitialPositionSet_RightBottom:=FALSE;
	Alarm_RightBottomMotorPos:=FALSE;
	Alarm_RightBottomMotorVelo:=FALSE;
ELSE
    //一点变动没有了，光栅异常，开始计时
    StableTimer_RightBottomLin(
        IN := TRUE,
        PT := LEHeartBeatAlarmTime,
        ET => StableTime_RightBottomLin
    );
	//记录电机初始位置，后后续对比做准备
	IF NOT IsInitialPositionSet_RightBottom THEN
        Pos_RightBottomMotor_Initial := Pos_RightBottomMotor;  // 记录初始位置
        IsInitialPositionSet_RightBottom := TRUE;
   	END_IF;
    
    // 100ms速度完全不变，开始监控电机速度和位置
    IF StableTimer_RightBottomLin.Q THEN
        Alarm_RightBottomLin := TRUE;  // 
			//电机位置对比及监测
			MotorPosChange_RightBottom:=ABS( Pos_RightBottomMotor-Pos_RightBottomMotor_Initial);
			IF MotorPosChange_RightBottom > Threshold_RightBottomMotorPos THEN
				Alarm_RightBottomMotorPos:=TRUE;
				ErrorID:=5007;
				ErrorDescription:='5007';
				Error:=TRUE;
				FB_PlcEmergencyStop();
				LED_Error:=TRUE;
			ELSE
				Alarm_RightBottomMotorPos:=FALSE;
			END_IF
			//电机速度监测
			IF Velo_RightBottomMotor > Threshold_RightBottomMotorVelo THEN
				Alarm_RightBottomMotorVelo:=TRUE;
				ErrorID:=5008;
				ErrorDescription:='5008';
				Error:=TRUE;
				FB_PlcEmergencyStop();
				LED_Error:=TRUE;
			ELSE
				Alarm_RightBottomMotorVelo:=FALSE;
			END_IF
    ELSE
        Alarm_RightBottomLin := FALSE;
	END_IF
END_IF
//PhaseUpper monitor
IF DeltaVelo_PhaseUpperLin > LEHeartBeatDeadZone THEN
    // 有变动，光栅正常，计数器归零，更新位置,重置所有状态
    StableTimer_PhaseUpperLin(IN := FALSE, PT := LEHeartBeatAlarmTime);
    Alarm_PhaseUpperLin := FALSE;
    Velo_PhaseUpperLin_Last := PhaseUpperLin.NcToPlc.ActVelo;  // 
    StableTime_PhaseUpperLin := T#0S;
	IsInitialPositionSet_PhaseUpper:=FALSE;
	Alarm_PhaseUpperMotorPos:=FALSE;
	Alarm_PhaseUpperMotorVelo:=FALSE;
ELSE
    //一点变动没有了，光栅异常，开始计时
    StableTimer_PhaseUpperLin(
        IN := TRUE,
        PT := LEHeartBeatAlarmTime,
        ET => StableTime_PhaseUpperLin
    );
	//记录电机初始位置，后后续对比做准备
	IF NOT IsInitialPositionSet_PhaseUpper THEN
        Pos_PhaseUpperMotor_Initial := Pos_PhaseUpperMotor;  // 记录初始位置
        IsInitialPositionSet_PhaseUpper := TRUE;
   	END_IF;
    
    // 100ms速度完全不变，开始监控电机速度和位置
    IF StableTimer_PhaseUpperLin.Q THEN
        Alarm_PhaseUpperLin := TRUE;  // 
			//电机位置对比及监测
			MotorPosChange_PhaseUpper:=ABS( Pos_PhaseUpperMotor-Pos_PhaseUpperMotor_Initial);
			IF MotorPosChange_PhaseUpper > Threshold_PhaseUpperMotorPos THEN
				Alarm_PhaseUpperMotorPos:=TRUE;
				ErrorID:=5009;
				ErrorDescription:='5009';
				Error:=TRUE;
				FB_PlcEmergencyStop();
				LED_Error:=TRUE;
			ELSE
				Alarm_PhaseUpperMotorPos:=FALSE;
			END_IF
			//电机速度监测
			IF Velo_PhaseUpperMotor > Threshold_PhaseUpperMotorVelo THEN
				Alarm_PhaseUpperMotorVelo:=TRUE;
				ErrorID:=5010;
				ErrorDescription:='5010';
				Error:=TRUE;
				FB_PlcEmergencyStop();
				LED_Error:=TRUE;
			ELSE
				Alarm_PhaseUpperMotorVelo:=FALSE;
			END_IF
    ELSE
        Alarm_PhaseUpperLin := FALSE;
	END_IF
END_IF
//PhaseLower monitor
IF DeltaVelo_PhaseLowerLin > LEHeartBeatDeadZone THEN
    // 有变动，光栅正常，计数器归零，更新位置,重置所有状态
    StableTimer_PhaseLowerLin(IN := FALSE, PT := LEHeartBeatAlarmTime);
    Alarm_PhaseLowerLin := FALSE;
    Velo_PhaseLowerLin_Last := PhaseLowerLin.NcToPlc.ActVelo;  // 
    StableTime_PhaseLowerLin := T#0S;
	IsInitialPositionSet_PhaseLower:=FALSE;
	Alarm_PhaseLowerMotorPos:=FALSE;
	Alarm_PhaseLowerMotorVelo:=FALSE;
ELSE
    //一点变动没有了，光栅异常，开始计时
    StableTimer_PhaseLowerLin(
        IN := TRUE,
        PT := LEHeartBeatAlarmTime,
        ET => StableTime_PhaseLowerLin
    );
	//记录电机初始位置，后后续对比做准备
	IF NOT IsInitialPositionSet_PhaseLower THEN
        Pos_PhaseLowerMotor_Initial := Pos_PhaseLowerMotor;  // 记录初始位置
        IsInitialPositionSet_PhaseLower := TRUE;
   	END_IF;
    
    // 100ms速度完全不变，开始监控电机速度和位置
    IF StableTimer_PhaseLowerLin.Q THEN
        Alarm_PhaseLowerLin := TRUE;  // 
			//电机位置对比及监测
			MotorPosChange_PhaseLower:=ABS( Pos_PhaseLowerMotor-Pos_PhaseLowerMotor_Initial);
			IF MotorPosChange_PhaseLower > Threshold_PhaseLowerMotorPos THEN
				Alarm_PhaseLowerMotorPos:=TRUE;
				ErrorID:=5011;
				ErrorDescription:='5011';
				Error:=TRUE;
				FB_PlcEmergencyStop();
				LED_Error:=TRUE;
			ELSE
				Alarm_PhaseLowerMotorPos:=FALSE;
			END_IF
			//电机速度监测
			IF Velo_PhaseLowerMotor > Threshold_PhaseLowerMotorVelo THEN
				Alarm_PhaseLowerMotorVelo:=TRUE;
				ErrorID:=5012;
				ErrorDescription:='5012';
				Error:=TRUE;
				FB_PlcEmergencyStop();
				LED_Error:=TRUE;
			ELSE
				Alarm_PhaseLowerMotorVelo:=FALSE;
			END_IF
    ELSE
        Alarm_PhaseLowerLin := FALSE;
	END_IF
END_IF
END_ACTION

ACTION A_LoadOpcIocShellExe:
R_TRIG_Exeload(CLK:=bExe_load_Prog, Q=> );
LoadOpcIocTON(PT:=T#10S);
CASE Exe_load_step OF
	0:
		LoadOpcIocTON.IN:=TRUE;
		IF R_TRIG_Exeload.Q THEN
			NT_StartProcess_Load.START:=FALSE;
			NT_StartProcess_Load.PATHSTR:='C:\HZB\OpcIocShell\IDControlIOC\startTwinCATOPCServer.bat';
			Exe_load_step:=10;
		END_IF;
	10:
		IF LoadOpcIocTON.Q THEN
			NT_StartProcess_Load.START:=TRUE;
			Exe_load_step:=20;
		END_IF
	20:
		LoadOpcIocTON.IN:=FALSE;
		IF NT_StartProcess_Load.ERR THEN
			Exe_load_step:=0;
		ELSE
			Exe_load_step:=30;
		END_IF;
	30:
		IF NOT NT_StartProcess_Load.BUSY THEN
			NT_StartProcess_Load.START:=FALSE;
			Exe_Load_Done:=TRUE;
			Exe_load_step:=0;
		END_IF;
END_CASE;

NT_StartProcess_Load(
	NETID:='' ,
	PATHSTR:= ,
	DIRNAME:= , 
	COMNDLINE:= , 
	START:= ,
	ERRID=> );
END_ACTION

ACTION A_MonitorMotorAndLE:
//Monitoring Motor and LE Position/Velocity
IF 	ABS(DeltaPos_LeftTop) > ThresholdDeltaPos_LeftTop THEN
	ErrorID:=6001;
	Error:=TRUE;
	ErrorDescription:='ABS(DeltaPos_LeftTop) > ThresholdDeltaPos_LeftTop';
	FB_PlcEmergencyStop();
	LED_Error:=TRUE;
END_IF
IF ABS(DeltaPos_RightTop) > ThresholdDeltaPos_RightTop THEN
	ErrorID:=6002;
	Error:=TRUE;
	ErrorDescription:='ABS(DeltaPos_RightTop) > ThresholdDeltaPos_RightTop';
	FB_PlcEmergencyStop();
	LED_Error:=TRUE;
END_IF
IF ABS(DeltaPos_LeftBottom) > ThresholdDeltaPos_LeftBottom THEN
	ErrorID:=6003;
	Error:=TRUE;
	ErrorDescription:='ABS(DeltaPos_LeftBottom) > ThresholdDeltaPos_LeftBottom';
	FB_PlcEmergencyStop();
	LED_Error:=TRUE;
END_IF
IF ABS(DeltaPos_RightBottom) > ThresholdDeltaPos_RightBottom THEN
	ErrorID:=6004;
	Error:=TRUE;
	ErrorDescription:='ABS(DeltaPos_RightBottom) > ThresholdDeltaPos_RightBottom';
	FB_PlcEmergencyStop();
	LED_Error:=TRUE;
END_IF
(*
IF ABS(DeltaPos_PhaseUpper) > ThresholdDeltaPos_PhaseUpper THEN
	ErrorID:=6005;
	Error:=TRUE;
	ErrorDescription:='ABS(DeltaPos_PhaseUpper) > ThresholdDeltaPos_PhaseUpper';
	FB_PlcEmergencyStop();
	LED_Error:=TRUE;
END_IF
IF ABS(DeltaPos_PhaseLower) > ThresholdDeltaPos_PhaseLower THEN
	ErrorID:=6006;
	Error:=TRUE;
	ErrorDescription:='ABS(DeltaPos_PhaseLower) > ThresholdDeltaPos_PhaseLower';
	FB_PlcEmergencyStop();
	LED_Error:=TRUE;
END_IF
*)
IF ABS(DeltaVelo_LeftTop) > ThresholdDeltaVelo_LeftTop THEN
	ErrorID:=6007;
	Error:=TRUE;
	ErrorDescription:='ABS(DeltaVelo_LeftTop) > ThresholdDeltaVelo_LeftTop';
	FB_PlcEmergencyStop();
	LED_Error:=TRUE;
END_IF
IF ABS(DeltaVelo_RightTop) > ThresholdDeltaVelo_RightTop THEN
	ErrorID:=6008;
	Error:=TRUE;
	ErrorDescription:='ABS(DeltaVelo_RightTop) > ThresholdDeltaVelo_RightTop';
	FB_PlcEmergencyStop();
	LED_Error:=TRUE;
END_IF
IF ABS(DeltaVelo_LeftBottom) > ThresholdDeltaVelo_LeftBottom THEN
	ErrorID:=6009;
	Error:=TRUE;
	ErrorDescription:='ABS(DeltaVelo_LeftBottom) > ThresholdDeltaVelo_LeftBottom';
	FB_PlcEmergencyStop();
	LED_Error:=TRUE;
END_IF
IF ABS(DeltaVelo_RightBottom) > ThresholdDeltaVelo_RightBottom THEN
	ErrorID:=6010;
	Error:=TRUE;
	ErrorDescription:='ABS(DeltaVelo_RightBottom) > ThresholdDeltaVelo_RightBottom';
	FB_PlcEmergencyStop();
	LED_Error:=TRUE;
END_IF
(*
IF ABS(DeltaVelo_PhaseUpper) > ThresholdDeltaVelo_PhaseUpper THEN
	ErrorID:=6011;
	Error:=TRUE;
	ErrorDescription:='ABS(DeltaVelo_PhaseUpper) > ThresholdDeltaVelo_PhaseUpper';
	FB_PlcEmergencyStop();
	LED_Error:=TRUE;
END_IF
IF ABS(DeltaVelo_PhaseLower) > ThresholdDeltaVelo_PhaseLower THEN
	ErrorID:=6012;
	Error:=TRUE;
	ErrorDescription:='ABS(DeltaVelo_PhaseLower) > ThresholdDeltaVelo_PhaseLower';
	FB_PlcEmergencyStop();
	LED_Error:=TRUE;
END_IF
*)
(*
//
//IF NotMoving ,Threshold is less
//
IF NOT moveStatusLeftTop THEN
		IF 	ABS(DeltaPos_LeftTop) > ThresholdDeltaPos_LeftTop/3 THEN
		ErrorID:=6009;
		Error:=TRUE;
		ErrorDescription:='ABS(DeltaPos_LeftTop) > ThresholdDeltaPos_LeftTop/3';
		FB_PlcEmergencyStop();
		LED_Error:=TRUE;
	END_IF
END_IF
IF NOT moveStatusRightTop THEN
	IF ABS(DeltaPos_RightTop) > ThresholdDeltaPos_RightTop/3 THEN
		ErrorID:=6010;
		Error:=TRUE;
		ErrorDescription:='ABS(DeltaPos_RightTop) > ThresholdDeltaPos_RightTop/3';
		FB_PlcEmergencyStop();
		LED_Error:=TRUE;
	END_IF
END_IF
IF NOT moveStatusLeftBottom THEN
	IF ABS(DeltaPos_LeftBottom) > ThresholdDeltaPos_LeftBottom/3 THEN
		ErrorID:=6011;
		Error:=TRUE;
		ErrorDescription:='ABS(DeltaPos_LeftBottom) > ThresholdDeltaPos_LeftBottom/3';
		FB_PlcEmergencyStop();
		LED_Error:=TRUE;
	END_IF
END_IF
IF NOT moveStatusRightBottom THEN
	IF ABS(DeltaPos_RightBottom) > ThresholdDeltaPos_RightBottom/3 THEN
		ErrorID:=6012;
		Error:=TRUE;
		ErrorDescription:='ABS(DeltaPos_RightBottom) > ThresholdDeltaPos_RightBottom';
		FB_PlcEmergencyStop();
		LED_Error:=TRUE;
	END_IF
END_IF

//
IF NOT moveStatusLeftTop THEN
	IF ABS(DeltaVelo_LeftTop) > ThresholdDeltaVelo_LeftTop/3 THEN
		ErrorID:=6013;
		Error:=TRUE;
		ErrorDescription:='ABS(DeltaVelo_LeftTop) > ThresholdDeltaVelo_LeftTop/3';
		FB_PlcEmergencyStop();
		LED_Error:=TRUE;
	END_IF
END_IF
IF NOT moveStatusRightTop THEN
	IF ABS(DeltaVelo_RightTop) > ThresholdDeltaVelo_RightTop/3 THEN
		ErrorID:=6014;
		Error:=TRUE;
		ErrorDescription:='ABS(DeltaVelo_RightTop) > ThresholdDeltaVelo_RightTop/3';
		FB_PlcEmergencyStop();
		LED_Error:=TRUE;
	END_IF
END_IF
IF NOT moveStatusLeftBottom THEN
	IF ABS(DeltaVelo_LeftBottom) > ThresholdDeltaVelo_LeftBottom/3 THEN
		ErrorID:=6015;
		Error:=TRUE;
		ErrorDescription:='ABS(DeltaVelo_LeftBottom) > ThresholdDeltaVelo_LeftBottom/3';
		FB_PlcEmergencyStop();
		LED_Error:=TRUE;
	END_IF
END_IF
IF NOT moveStatusRightBottom THEN
	IF ABS(DeltaVelo_RightBottom) > ThresholdDeltaVelo_RightBottom/3 THEN
		ErrorID:=6016;
		Error:=TRUE;
		ErrorDescription:='ABS(DeltaVelo_RightBottom) > ThresholdDeltaVelo_RightBottom/3';
		FB_PlcEmergencyStop();
		LED_Error:=TRUE;
	END_IF
END_IF
*)
END_ACTION

ACTION A_PolarStatus:
// 调用
fbPolar(
    Pos_PhaseUpper := Pos_PhaseUpperLin,
    Pos_PhaseLower := Pos_PhaseLowerLin,
    Upper_HM  := stPolarizationParam.Upper_HM,
    Lower_HM  := stPolarizationParam.Lower_HM,
    Upper_VM1 := stPolarizationParam.Upper_VM1,
    Lower_VM1 := stPolarizationParam.Lower_VM1,
    Upper_VM2 := stPolarizationParam.Upper_VM2,
    Lower_VM2 := stPolarizationParam.Lower_VM2,
    Upper_LC  := stPolarizationParam.Upper_LC,
    Lower_LC  := stPolarizationParam.Lower_LC,
    Upper_RC  := stPolarizationParam.Upper_RC,
    Lower_RC  := stPolarizationParam.Lower_RC,
    rTolerance := stPolarizationParam.Tolerance
);
END_ACTION

ACTION A_PosDiffDetectiion:
IF ABS(PosDiff_LeftTopLin_actual)>PosDiff_LeftTopLin THEN
	ErrorID:=201;
	Error:=TRUE;
	ErrorDescription:='ABS(PosDiff_LeftTopLin_actual)>PosDiff_LeftTopLin';
	FB_PlcEmergencyStop();
	LED_Error:=TRUE;
END_IF
IF ABS(PosDiff_RightTopLin_actual)>PosDiff_RightTopLin THEN
	ErrorID:=202;
	Error:=TRUE;
	ErrorDescription:='ABS(PosDiff_RightTopLin_actual)>PosDiff_RightTopLin';
	FB_PlcEmergencyStop();
	LED_Error:=TRUE;
END_IF
IF ABS(PosDiff_LeftBottomLin_actual)>PosDiff_LeftBottomLin THEN
	ErrorID:=203;
	Error:=TRUE;
	ErrorDescription:='ABS(PosDiff_LeftBottomLin_actual)>PosDiff_LeftBottomLin';
	FB_PlcEmergencyStop();
	LED_Error:=TRUE;
END_IF
IF ABS(PosDiff_RightBottomLin_actual)>PosDiff_RightBottomLin THEN
	ErrorID:=204;
	ErrorDescription:='ABS(PosDiff_RightBottomLin_actual)>PosDiff_RightBottomLin';
	Error:=TRUE;
	FB_PlcEmergencyStop();
	LED_Error:=TRUE;
END_IF
IF ABS(PosDiff_PhaseUpperLin_actual)>PosDiff_PhaseUpperLin THEN
	ErrorID:=205;
	Error:=TRUE;
	ErrorDescription:='ABS(PosDiff_PhaseUpperLin_actual)>PosDiff_PhaseUpperLin';
	FB_PlcEmergencyStop();
	LED_Error:=TRUE;
END_IF
IF ABS(PosDiff_PhaseLowerLin_actual)>PosDiff_PhaseLowerLin THEN
	ErrorID:=206;
	ErrorDescription:='ABS(PosDiff_PhaseLowerLin_actual)>PosDiff_PhaseLowerLin';
	Error:=TRUE;
	FB_PlcEmergencyStop();
	LED_Error:=TRUE;
END_IF
//
IF ABS(PosDiff_LeftTopLin_actual-PosDiff_RightTopLin_actual)>0.05 THEN
	ErrorID:=207;
	ErrorDescription:='ABS(PosDiff_LeftTopLin_actual-PosDiff_RightTopLin_actual)>0.05';
	Error:=TRUE;
	FB_PlcEmergencyStop();
	LED_Error:=TRUE;
ELSIF ABS(PosDiff_LeftBottomLin_actual-PosDiff_RightBottomLin_actual)>0.05 THEN
	ErrorID:=28;
	ErrorDescription:='ABS(PosDiff_LeftBottomLin_actual-PosDiff_RightBottomLin_actual)>0.05';
	Error:=TRUE;
	FB_PlcEmergencyStop();
	LED_Error:=TRUE;
END_IF
END_ACTION

ACTION A_RestartDrivers:
Relay_EL2624[0]:=btn_RestartDriver1;
Relay_EL2624[1]:=btn_RestartDriver2;
Relay_EL2624[2]:=btn_RestartDriver3;
Relay_EL2624[3]:=btn_RestartDriver4;
Relay_EL2624[4]:=btn_RestartDriver5;
Relay_EL2624[5]:=btn_RestartDriver6;
Relay_EL2624[6]:=btn_RestartDriver7;
Relay_EL2624[7]:=btn_RestartDriver8;
///
//1.上升沿触发，btn_RestartDrivers上升沿后，btn_RestartDriver1~8全部高电平
//2、3s后，Driver1~8全部恢复低电平
//3、恢复全部状态到初始
///
RestartDriver_RTRIG(CLK:=btn_RestartDriversAll);
IF RestartDriver_RTRIG.Q THEN
	RestartDriver_Triggered:=TRUE;
	RestartDriver_Done:=FALSE;
END_IF
IF RestartDriver_Triggered THEN
	CASE RestartDriver_State OF
		0:
			btn_RestartDriver1:=TRUE;
			btn_RestartDriver2:=TRUE;
			btn_RestartDriver3:=TRUE;
			btn_RestartDriver4:=TRUE;
			btn_RestartDriver5:=TRUE;
			btn_RestartDriver6:=TRUE;
			btn_RestartDriver7:=TRUE;
			btn_RestartDriver8:=TRUE;
			//计时开始
			RestartDriver_TON(PT:=T#10S);
			RestartDriver_TON.IN:=TRUE;
			IF RestartDriver_TON.Q THEN
				RestartDriver_State:=1;
			END_IF
		1:
			btn_RestartDriver1:=FALSE;
			btn_RestartDriver2:=FALSE;
			btn_RestartDriver3:=FALSE;
			btn_RestartDriver4:=FALSE;
			btn_RestartDriver5:=FALSE;
			btn_RestartDriver6:=FALSE;
			btn_RestartDriver7:=FALSE;
			btn_RestartDriver8:=FALSE;
			RestartDriver_State:=88;
		88:
			RestartDriver_TON.IN:=FALSE;
			btn_RestartDriversAll:=FALSE;
			RestartDriver_State:=0;
			RestartDriver_Triggered:=FALSE;
			RestartDriver_Done:=TRUE;
	END_CASE
END_IF
END_ACTION

ACTION A_RestartTC:
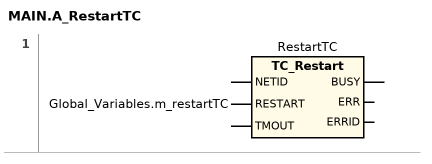
// NETWORK 1
RestartTC(RESTART := Global_Variables.m_restartTC); // TC_Restart
END_ACTION

ACTION A_SafePlcStartInit:
fb_ton0(PT:=t#1s);
fb_ton1(PT:=t#0.1s);
fb_ton2(PT:=t#0.1s);
fb_ton3(PT:=t#0.1s);

CASE SafeStatus OF
	0:
		IF COM_ERROR OR NOT Estop_Out THEN
			Err_Ack:=TRUE;
			fb_ton0.IN:=TRUE;
			SafeStatus:=1;
		ELSE
			SafePLCRunOK:=TRUE;
			SafeStatus:=0;
		END_IF
	1:
		IF fb_ton0.Q THEN
			Err_Ack:=FALSE;
			Safe_run:=TRUE;
			fb_ton1.IN:=TRUE;
			SafeStatus:=2;
		END_IF

	2:
		IF fb_ton1.Q THEN
			IF Estop_RunAndRestart=FALSE THEN
				Estop_RunAndRestart:=TRUE;
				fb_ton2.IN:=TRUE;
				SafeStatus:=3;
			END_IF
		END_IF
	3:
		IF fb_ton2.Q THEN
			IF Estop_RunAndRestart THEN
				Estop_RunAndRestart:=FALSE;
				fb_ton3.IN:=TRUE;
				SafeStatus:=4;
			END_IF
		END_IF
	4:
		IF fb_ton3.Q THEN
			IF Estop_Out THEN
				SafePLCRunOK:=TRUE;
				SafeStatus:=0;
			ELSE
				SafePLCRunOK:=FALSE;
				//Error:=TRUE;
				//ErrorId:=301;
				//ErrorDescription:='SafePLCRunOK fail';
			END_IF
		fb_ton0.IN:=FALSE;
		fb_ton1.IN:=FALSE;
		fb_ton2.IN:=FALSE;
		fb_ton3.IN:=FALSE;
		END_IF


END_CASE
END_ACTION

ACTION A_SetAxisPosition:
fb_ton4(PT:=t#0.5s);
CASE SetAxisPosState OF
	0:	(*FB_Set_AxisPosition*)
		FB_Set_AxisPosition(Execute:=TRUE);
		fb_ton4.IN:=TRUE;
		SetAxisPosState:=1;
	1:	(*wait*)
		FB_Set_AxisPosition();
		IF NOT FB_Set_AxisPosition.Done THEN		(*FB_Set_AxisPositionÃ»ÓÐÖ´ÐÐÍê£¬wait£¬³¬Ê±FB Error*)
			IF NOT fb_ton4.Q THEN
				SetAxisPosState:=1;
			ELSE
				SetAxisPosState:=99;
			END_IF
		ELSE
			SetAxisPosState:=88;
		END_IF
	88:
		SetAxisPosState:=0;
		SetAxisPositionDone:=TRUE;
		Error:=FALSE;
		ErrorID:=0;
		FB_Set_AxisPosition.Execute:=FALSE;
		fb_ton4.IN:=FALSE;
	99:
		SetAxisPosState:=99;
		SetAxisPositionDone:=FALSE;
		Error:=TRUE;
		FB_Set_AxisPosition.Execute:=FALSE;
		fb_ton4.IN:=FALSE;
		LED_Error:=TRUE;
		ErrorID:=401;
		ErrorDescription:='SetAxisPosition fail';
END_CASE
END_ACTION

ACTION A_SetLinearEncoderPositionBias:
//设置bias开始
A_SetLinearEncoderPositionBiasMC();
PositionBiasTON(PT:=T#0.1S);
CASE state_setLEPosBias OF
	0:
		PositionBiasTON.IN:=TRUE;
		IF MC_SetLEPosBias_LeftTop.Error OR MC_SetLEPosBias_RightTop.Error OR 
			MC_SetLEPosBias_LeftBottom.Error OR MC_SetLEPosBias_RightBottom.Error OR
			MC_SetLEPosBias_PhaseUpper.Error OR MC_SetLEPosBias_PhaseLower.Error THEN
			state_setLEPosBias:=-100;
		ELSE 
			state_setLEPosBias:=1;
		END_IF
	1:
		IF NOT MC_SetLEPosBias_LeftTop.Done OR NOT MC_SetLEPosBias_RightTop.Done OR 
			NOT MC_SetLEPosBias_LeftBottom.Done OR NOT MC_SetLEPosBias_RightBottom.Done OR
			NOT MC_SetLEPosBias_PhaseUpper.Done OR NOT MC_SetLEPosBias_PhaseLower.Done  THEN
			MC_SetLEPosBias_LeftTop.Execute:=TRUE;
			MC_SetLEPosBias_RightTop.Execute:=TRUE;
			MC_SetLEPosBias_LeftBottom.Execute:=TRUE;
			MC_SetLEPosBias_RightBottom.Execute:=TRUE;
			MC_SetLEPosBias_PhaseUpper.Execute:=TRUE;
			MC_SetLEPosBias_PhaseLower.Execute:=TRUE;
			state_setLEPosBias:=2;
		ELSE
			state_setLEPosBias:=-100;
		END_IF
	2:
		IF NOT MC_SetLEPosBias_LeftTop.Done OR NOT MC_SetLEPosBias_RightTop.Done OR 
			NOT MC_SetLEPosBias_LeftBottom.Done OR NOT MC_SetLEPosBias_RightBottom.Done OR
			NOT MC_SetLEPosBias_PhaseUpper.Done OR NOT MC_SetLEPosBias_PhaseLower.Done THEN
			IF NOT PositionBiasTON.Q THEN
				state_setLEPosBias:=2;
			ELSE
				state_setLEPosBias:=-100;
			END_IF
		END_IF
		IF  MC_SetLEPosBias_LeftTop.Done AND MC_SetLEPosBias_RightTop.Done AND
			MC_SetLEPosBias_LeftBottom.Done AND MC_SetLEPosBias_RightBottom.Done AND
			MC_SetLEPosBias_PhaseUpper.Done AND MC_SetLEPosBias_PhaseLower.Done THEN
			state_setLEPosBias:=88;
		END_IF	
		IF MC_SetLEPosBias_LeftTop.Error OR MC_SetLEPosBias_RightTop.Error OR 
			MC_SetLEPosBias_LeftBottom.Error OR MC_SetLEPosBias_RightBottom.Error OR
			MC_SetLEPosBias_PhaseUpper.Error OR MC_SetLEPosBias_PhaseLower.Error THEN
			state_setLEPosBias:=-100;
		END_IF 
		
	88:
		PositionBiasTON.IN:=FALSE;
		PositionBiasDone:=TRUE;
	-100:
		PositionBiasTON.IN:=FALSE;
		PositionBiasDone:=FALSE;
		Error:=TRUE;
		ErrorId:=901;
		ErrorDescription:='Set LinearEncoderPositionBias Error';
		Plc_EmergencyStop:=FALSE;
END_CASE
END_ACTION

ACTION A_SetLinearEncoderPositionBiasMC:
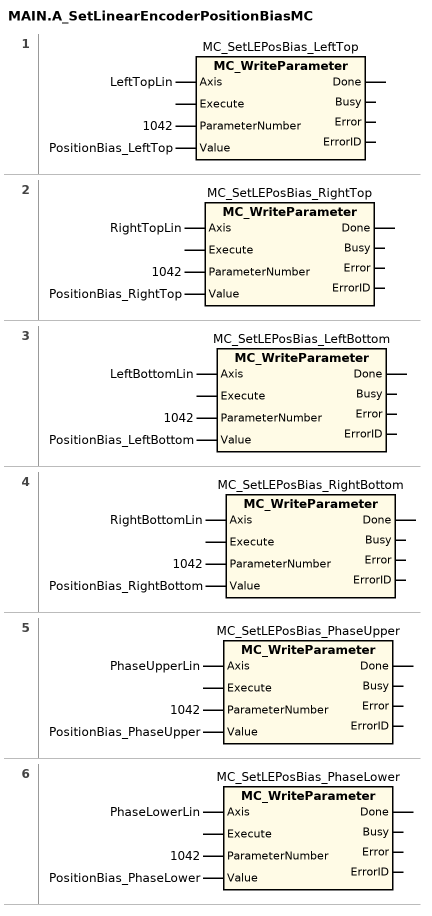
// NETWORK 1
MC_SetLEPosBias_LeftTop(Axis := LeftTopLin, ParameterNumber := 1042, Value := PositionBias_LeftTop); // MC_WriteParameter

// NETWORK 2
MC_SetLEPosBias_RightTop(Axis := RightTopLin, ParameterNumber := 1042, Value := PositionBias_RightTop); // MC_WriteParameter

// NETWORK 3
MC_SetLEPosBias_LeftBottom(Axis := LeftBottomLin, ParameterNumber := 1042, Value := PositionBias_LeftBottom); // MC_WriteParameter

// NETWORK 4
MC_SetLEPosBias_RightBottom(
    Axis := RightBottomLin,
    ParameterNumber := 1042,
    Value := PositionBias_RightBottom); // MC_WriteParameter

// NETWORK 5
MC_SetLEPosBias_PhaseUpper(Axis := PhaseUpperLin, ParameterNumber := 1042, Value := PositionBias_PhaseUpper); // MC_WriteParameter

// NETWORK 6
MC_SetLEPosBias_PhaseLower(Axis := PhaseLowerLin, ParameterNumber := 1042, Value := PositionBias_PhaseLower); // MC_WriteParameter
END_ACTION

ACTION A_SetMotorAxisPosition:
fb_ton4_2(PT:=T#0.5S);
CASE SetMotorAxisPosState OF
	0:	(*FB_Set_AxisPosition*)
		FB_Set_MotorAxisPosition(Execute:=TRUE);
		fb_ton4_2.IN:=TRUE;
		SetMotorAxisPosState:=1;
	1:	(*wait*)
		FB_Set_MotorAxisPosition();
		IF NOT FB_Set_MotorAxisPosition.Done THEN		
			IF NOT fb_ton4_2.Q THEN
				SetMotorAxisPosState:=1;
			ELSE
				SetMotorAxisPosState:=99;
			END_IF
		ELSE
			SetMotorAxisPosState:=88;
		END_IF
	88:
		SetMotorAxisPosState:=0;
		SetMotorAxisPositionDone:=TRUE;
		Error:=FALSE;
		ErrorID:=0;
		FB_Set_MotorAxisPosition.Execute:=FALSE;
		fb_ton4_2.IN:=FALSE;
	99:
		SetMotorAxisPosState:=99;
		SetMotorAxisPositionDone:=FALSE;
		Error:=TRUE;
		FB_Set_MotorAxisPosition.Execute:=FALSE;
		fb_ton4_2.IN:=FALSE;
		LED_Error:=TRUE;
		ErrorID:=401;
		ErrorDescription:='SetMotorAxisPosition fail';
END_CASE
END_ACTION

ACTION A_SetPhaseLowerAxisPosition:
fb_ton8(PT:=T#0.5S);
CASE SetPhaseLowerAxisPosState OF
	0:	(*FB_Set_PhaseLowerAxisPosition*)
		FB_Set_PhaseLowerAxisPosition(Execute:=TRUE);
		fb_ton8.IN:=TRUE;
		SetPhaseLowerAxisPosState:=1;
	1:	(*wait*)
		FB_Set_PhaseLowerAxisPosition();
		IF NOT FB_Set_PhaseLowerAxisPosition.Done THEN		(*FB_Set_AxisPositionÃ»ÓÐÖ´ÐÐÍê£¬wait£¬³¬Ê±FB Error*)
			IF NOT fb_ton8.Q THEN
				SetPhaseLowerAxisPosState:=1;
			ELSE
				SetPhaseLowerAxisPosState:=99;
			END_IF
		ELSE
			SetPhaseLowerAxisPosState:=88;
		END_IF
	88:
		SetPhaseLowerAxisPosState:=0;
		SetPhaseLowerAxisPositionDone:=TRUE;
		Error:=FALSE;
		ErrorID:=0;
		FB_Set_PhaseLowerAxisPosition.Execute:=FALSE;
		fb_ton8.IN:=FALSE;
	99:
		SetPhaseLowerAxisPosState:=99;
		SetPhaseLowerAxisPositionDone:=FALSE;
		Error:=TRUE;
		FB_Set_PhaseLowerAxisPosition.Execute:=FALSE;
		fb_ton8.IN:=FALSE;
		LED_Error:=TRUE;
		ErrorID:=403;
		ErrorDescription:='SetPhaseLowerAxisPosition fail';
END_CASE
END_ACTION

ACTION A_SetPhaseLowerMotorAxisPosition:
fb_ton8_2(PT:=T#0.5S);
CASE SetPhaseLowerMotorAxisPosState OF
	0:	(*FB_Set_PhaseLowerMotorAxisPosition*)
		FB_Set_PhaseLowerMotorAxisPosition(Execute:=TRUE);
		fb_ton8_2.IN:=TRUE;
		SetPhaseLowerMotorAxisPosState:=1;
	1:	(*wait*)
		FB_Set_PhaseLowerMotorAxisPosition();
		IF NOT FB_Set_PhaseLowerMotorAxisPosition.Done THEN		(*FB_Set_AxisPositionÃ»ÓÐÖ´ÐÐÍê£¬wait£¬³¬Ê±FB Error*)
			IF NOT fb_ton8_2.Q THEN
				SetPhaseLowerMotorAxisPosState:=1;
			ELSE
				SetPhaseLowerMotorAxisPosState:=99;
			END_IF
		ELSE
			SetPhaseLowerMotorAxisPosState:=88;
		END_IF
	88:
		SetPhaseLowerMotorAxisPosState:=0;
		SetPhaseLowerMotorAxisPositionDone:=TRUE;
		Error:=FALSE;
		ErrorID:=0;
		FB_Set_PhaseLowerMotorAxisPosition.Execute:=FALSE;
		fb_ton8_2.IN:=FALSE;
	99:
		SetPhaseLowerMotorAxisPosState:=99;
		SetPhaseLowerMotorAxisPositionDone:=FALSE;
		Error:=TRUE;
		FB_Set_PhaseLowerMotorAxisPosition.Execute:=FALSE;
		fb_ton8_2.IN:=FALSE;
		LED_Error:=TRUE;
		ErrorID:=403;
		ErrorDescription:='SetPhaseLowerMotorAxisPosition fail';
END_CASE
END_ACTION

ACTION A_SetPhaseUpperAxisPosition:
fb_ton7(PT:=T#0.5S);
CASE SetPhaseUpperAxisPosState OF
	0:	(*FB_Set_PhaseUpperAxisPosition*)
		FB_Set_PhaseUpperAxisPosition(Execute:=TRUE);
		fb_ton7.IN:=TRUE;
		SetPhaseUpperAxisPosState:=1;
	1:	(*wait*)
		FB_Set_PhaseUpperAxisPosition();
		IF NOT FB_Set_PhaseUpperAxisPosition.Done THEN		(*FB_Set_AxisPositionÃ»ÓÐÖ´ÐÐÍê£¬wait£¬³¬Ê±FB Error*)
			IF NOT fb_ton7.Q THEN
				SetPhaseUpperAxisPosState:=1;
			ELSE
				SetPhaseUpperAxisPosState:=99;
			END_IF
		ELSE
			SetPhaseUpperAxisPosState:=88;
		END_IF
	88:
		SetPhaseUpperAxisPosState:=0;
		SetPhaseUpperAxisPositionDone:=TRUE;
		Error:=FALSE;
		ErrorID:=0;
		FB_Set_PhaseUpperAxisPosition.Execute:=FALSE;
		fb_ton7.IN:=FALSE;
	99:
		SetPhaseUpperAxisPosState:=99;
		SetPhaseUpperAxisPositionDone:=FALSE;
		Error:=TRUE;
		FB_Set_PhaseUpperAxisPosition.Execute:=FALSE;
		fb_ton7.IN:=FALSE;
		LED_Error:=TRUE;
		ErrorID:=402;
		ErrorDescription:='SetPhaseUpperAxisPosition fail';
END_CASE
END_ACTION

ACTION A_SetPhaseUpperMotorAxisPosition:
fb_ton7_2(PT:=T#0.5S);
CASE SetPhaseUpperMotorAxisPosState OF
	0:	(*FB_Set_PhaseUpperAxisPosition*)
		FB_Set_PhaseUpperMotorAxisPosition(Execute:=TRUE);
		fb_ton7_2.IN:=TRUE;
		SetPhaseUpperMotorAxisPosState:=1;
	1:	(*wait*)
		FB_Set_PhaseUpperMotorAxisPosition();
		IF NOT FB_Set_PhaseUpperMotorAxisPosition.Done THEN		(*FB_Set_AxisPositionÃ»ÓÐÖ´ÐÐÍê£¬wait£¬³¬Ê±FB Error*)
			IF NOT fb_ton7_2.Q THEN
				SetPhaseUpperMotorAxisPosState:=1;
			ELSE
				SetPhaseUpperMotorAxisPosState:=99;
			END_IF
		ELSE
			SetPhaseUpperMotorAxisPosState:=88;
		END_IF
	88:
		SetPhaseUpperMotorAxisPosState:=0;
		SetPhaseUpperMotorAxisPositionDone:=TRUE;
		Error:=FALSE;
		ErrorID:=0;
		FB_Set_PhaseUpperMotorAxisPosition.Execute:=FALSE;
		fb_ton7_2.IN:=FALSE;
	99:
		SetPhaseUpperMotorAxisPosState:=99;
		SetPhaseUpperMotorAxisPositionDone:=FALSE;
		Error:=TRUE;
		FB_Set_PhaseUpperMotorAxisPosition.Execute:=FALSE;
		fb_ton7_2.IN:=FALSE;
		LED_Error:=TRUE;
		ErrorID:=402;
		ErrorDescription:='SetPhaseUpperMotorAxisPosition fail';
END_CASE
END_ACTION

END_PROGRAM

(* stored: Version 1.1.0.1, ProductVersion 3.1.4024.6
   POU MAIN: Id {9221b602-3f7e-4757-b581-54b56182ad8f}, SpecialFunc None
   Folder Axis: Id {3eb3b5b7-a5d5-4d06-be7c-05e13125e510}
   Folder Check: Id {010fabb8-e18f-4120-a985-758e6fd55448}
   Folder Driver: Id {4350ce85-0586-4023-bc46-2cdffd7a9c8a}
   Folder LinearEncoder: Id {059dd61e-7778-40dc-bb8d-282e70434fee}
   Folder PolarStatus: Id {96dd34fe-4e07-41f6-b5de-0b051764b39b}
   Folder Recipe: Id {b4cf8559-847d-478e-99d6-23420c56f08c}
   Folder Safe: Id {05d14914-bd26-4aa9-9f6b-59a79d201008}
   Folder TC: Id {241a329f-2cca-4424-8363-173b04696ef4}
   Folder Temperature: Id {208f15b3-de64-4bc9-957f-ed1bc6c64ee5}
   Action A_CheckHardwareEmergencyStopStatus: Id {c59a955b-0a8f-43a7-a0e7-3ab11b3d5ab6}
   Action A_CheckKillSwitch: Id {158eed83-fba1-4051-b569-3585448d2a5a}
   Action A_CheckLimitSwitch: Id {1026ae85-58e3-4004-8dd3-becfab0085f9}
   Action A_CheckLinearEncoder: Id {04ef6a41-e2ba-498d-aa00-f823237bb5de}
   Action A_CheckMaxVelocity: Id {b95fb694-2a75-4423-bee6-d704fd7332fe}
   Action A_GetDriverStatus: Id {e05cf975-7b3e-4430-bb2e-a308f4391f1b}
   Action A_GetDriverStatusMC: Id {2d8972a4-2924-4445-a68a-757b585b0760}
   Action A_GetMotorTemperature: Id {177f6aa7-fb59-4f66-a7a6-1b4260347e60}
   Action A_GetTemperatureSensorsData: Id {d73fb87c-9e06-4b36-8cf6-68d5032eab30}
   Action A_InitAxisParameters: Id {a92c2dd6-12b0-4a71-a4bc-d7afbc965cb4}
   Action A_InitRecipeParameters: Id {6aa76980-7ae7-46e7-9688-f94b6fa6510d}
   Action A_KillOpcIocShellExe: Id {e0252576-ad9e-49ed-bcc5-7f64aacd5ffe}
   Action A_LEHeartBeatMonitor: Id {c15e81d3-3944-4229-9ecc-53c2921ba7f3}
   Action A_LoadOpcIocShellExe: Id {e69e9ea4-205f-45b3-85e7-e1c1b3150dfb}
   Action A_MonitorMotorAndLE: Id {8906040e-6c25-4137-b340-4fb081d521ce}
   Action A_PolarStatus: Id {b051506f-50a1-4381-9f89-0ba3c08f64b3}
   Action A_PosDiffDetectiion: Id {e857c546-d367-4f19-9434-ed29c144eb6f}
   Action A_RestartDrivers: Id {d1732994-27d5-4d0a-bd2e-fb077b65c9a9}
   Action A_RestartTC: Id {737d9420-c364-46ec-805e-ce283c214994}
   Action A_SafePlcStartInit: Id {4d1a8480-9923-4117-8ca7-ea613a82dfad}
   Action A_SetAxisPosition: Id {eb32aedd-8f01-44b1-96a9-73f233ea8548}
   Action A_SetLinearEncoderPositionBias: Id {6f3d3f8e-255d-4e09-853f-5fdf91122229}
   Action A_SetLinearEncoderPositionBiasMC: Id {d950edd3-252b-4c3c-9e26-a84e2707fa62}
   Action A_SetMotorAxisPosition: Id {1f7b7b3c-5e38-4a99-82a4-a1df4bf05d0c}
   Action A_SetPhaseLowerAxisPosition: Id {1fc13eaf-295a-4edf-80b0-8f2b92a70814}
   Action A_SetPhaseLowerMotorAxisPosition: Id {35e44bf9-a305-4255-8e2b-9610d7f39351}
   Action A_SetPhaseUpperAxisPosition: Id {e7a3e71e-f61e-4035-868f-571222f71b87}
   Action A_SetPhaseUpperMotorAxisPosition: Id {1a024de9-c34c-4374-9903-8d686c5a4886} *)
